LIN {X 0,Y 425.295,Z 309.51,A -85,B 0,C 180,E1 20716.386,E2 20716.386} C_VEL
LIN {X 0,Y 425.304,Z 309.491,A -85,B 0,C 180,E1 20712.629,E2 20712.629} C_VEL
LIN {X 0,Y 425.291,Z 309.491,A -85,B 0,C 180,E1 20708.79,E2 20708.79} C_VEL
LIN {X 0,Y 425.259,Z 309.512,A -85,B 0,C 180,E1 20705.126,E2 20705.126} C_VEL
LIN {X 0,Y 425.246,Z 309.506,A -85,B 0,C 180,E1 20701.347,E2 20701.347} C_VEL
LIN {X 0,Y 425.238,Z 309.495,A -85,B 0,C 180,E1 20697.574,E2 20697.574} C_VEL
LIN {X 0,Y 425.253,Z 309.511,A -85,B 0,C 180,E1 20693.791,E2 20693.791} C_VEL
LIN {X 0,Y 425.279,Z 309.498,A -85,B 0,C 180,E1 20690.086,E2 20690.086} C_VEL
LIN {X 0,Y 425.305,Z 309.487,A -85,B 0,C 180,E1 20686.264,E2 20686.264} C_VEL
LIN {X 0,Y 425.294,Z 309.508,A -85,B 0,C 180,E1 20682.486,E2 20682.486} C_VEL
LIN {X 0,Y 425.275,Z 309.503,A -85,B 0,C 180,E1 20678.772,E2 20678.772} C_VEL
LIN {X 0,Y 425.262,Z 309.492,A -85,B 0,C 180,E1 20675.111,E2 20675.111} C_VEL
LIN {X 0,Y 425.268,Z 309.502,A -85,B 0,C 180,E1 20671.276,E2 20671.276} C_VEL
LIN {X 0,Y 425.284,Z 309.507,A -85,B 0,C 180,E1 20667.565,E2 20667.565} C_VEL
LIN {X 0,Y 425.308,Z 309.508,A -85,B 0,C 180,E1 20663.837,E2 20663.837} C_VEL
LIN {X 0,Y 425.328,Z 309.506,A -85,B 0,C 180,E1 20660.026,E2 20660.026} C_VEL
LIN {X 0,Y 425.318,Z 309.499,A -85,B 0,C 180,E1 20656.092,E2 20656.092} C_VEL
LIN {X 0,Y 425.311,Z 309.478,A -85,B 0,C 180,E1 20652.223,E2 20652.223} C_VEL
LIN {X 0,Y 425.322,Z 309.731,A -85,B 0,C 180,E1 20648.704,E2 20648.704} C_VEL
LIN {X 0,Y 431.316,Z 325.075,A -85,B 0,C 180,E1 20645.907,E2 20645.907} C_VEL
LIN {X 0,Y 437.334,Z 341.625,A -85,B 0,C 180,E1 20643.199,E2 20643.199} C_VEL
LIN {X 0,Y 438.46,Z 344.163,A -85,B 0,C 180,E1 20642.946,E2 20642.946} C_VEL
LIN {X 0,Y 445.18,Z 356.721,A -85,B 0,C 180,E1 20642.081,E2 20642.081} C_VEL
LIN {X 0,Y 447.01,Z 366.68,A -85,B 0,C 180,E1 20641.733,E2 20641.733} C_VEL
LIN {X 0,Y 443.897,Z 554.794,A -85,B 0,C 180,E1 20638.73,E2 20638.73} C_VEL
LIN {X 0,Y 442.939,Z 562.472,A -85,B 0,C 180,E1 20638.628,E2 20638.628} C_VEL
LIN {X 0,Y 437.427,Z 580.609,A -85,B 0,C 180,E1 20638.46,E2 20638.46} C_VEL
LIN {X 0,Y 435.926,Z 588.027,A -85,B 0,C 180,E1 20638.239,E2 20638.239} C_VEL
LIN {X 0,Y 435.833,Z 589.062,A -85,B 0,C 180,E1 20638.193,E2 20638.193} C_VEL
LIN {X 0,Y 434.586,Z 606.139,A -85,B 0,C 180,E1 20637.321,E2 20637.321} C_VEL
LIN {X 0,Y 432.916,Z 623.479,A -85,B 0,C 180,E1 20636.175,E2 20636.175} C_VEL
LIN {X 0,Y 430.996,Z 639.731,A -85,B 0,C 180,E1 20634.827,E2 20634.827} C_VEL
LIN {X 0,Y 428.968,Z 654.603,A -85,B 0,C 180,E1 20633.313,E2 20633.313} C_VEL
LIN {X 0,Y 426.86,Z 668.614,A -85,B 0,C 180,E1 20631.576,E2 20631.576} C_VEL
LIN {X 0,Y 424.795,Z 681.338,A -85,B 0,C 180,E1 20629.668,E2 20629.668} C_VEL
LIN {X 0,Y 422.892,Z 692.644,A -85,B 0,C 180,E1 20627.615,E2 20627.615} C_VEL
LIN {X 0,Y 421.141,Z 703.114,A -85,B 0,C 180,E1 20625.279,E2 20625.279} C_VEL
LIN {X 0,Y 419.749,Z 711.572,A -85,B 0,C 180,E1 20622.939,E2 20622.939} C_VEL
LIN {X 0,Y 418.624,Z 718.946,A -85,B 0,C 180,E1 20620.319,E2 20620.319} C_VEL
LIN {X 0,Y 417.88,Z 724.436,A -85,B 0,C 180,E1 20617.7,E2 20617.7} C_VEL
LIN {X 0,Y 417.414,Z 728.221,A -85,B 0,C 180,E1 20615.085,E2 20615.085} C_VEL
LIN {X 0,Y 417.168,Z 730.486,A -85,B 0,C 180,E1 20612.335,E2 20612.335} C_VEL
LIN {X 0,Y 417.109,Z 731.085,A -85,B 0,C 180,E1 20609.588,E2 20609.588} C_VEL
LIN {X 0,Y 417.21,Z 730.043,A -85,B 0,C 180,E1 20606.84,E2 20606.84} C_VEL
LIN {X 0,Y 417.516,Z 727.312,A -85,B 0,C 180,E1 20604.09,E2 20604.09} C_VEL
LIN {X 0,Y 418.1,Z 722.784,A -85,B 0,C 180,E1 20601.335,E2 20601.335} C_VEL
LIN {X 0,Y 418.949,Z 716.685,A -85,B 0,C 180,E1 20598.715,E2 20598.715} C_VEL
LIN {X 0,Y 420.139,Z 709.085,A -85,B 0,C 180,E1 20596.233,E2 20596.233} C_VEL
LIN {X 0,Y 421.646,Z 700.029,A -85,B 0,C 180,E1 20593.893,E2 20593.893} C_VEL
LIN {X 0,Y 423.426,Z 689.42,A -85,B 0,C 180,E1 20591.672,E2 20591.672} C_VEL
LIN {X 0,Y 425.411,Z 677.603,A -85,B 0,C 180,E1 20589.645,E2 20589.645} C_VEL
LIN {X 0,Y 427.552,Z 664.114,A -85,B 0,C 180,E1 20587.738,E2 20587.738} C_VEL
LIN {X 0,Y 429.701,Z 649.518,A -85,B 0,C 180,E1 20586.045,E2 20586.045} C_VEL
LIN {X 0,Y 431.738,Z 633.856,A -85,B 0,C 180,E1 20584.559,E2 20584.559} C_VEL
LIN {X 0,Y 433.596,Z 617.11,A -85,B 0,C 180,E1 20583.279,E2 20583.279} C_VEL
LIN {X 0,Y 435.079,Z 600.265,A -85,B 0,C 180,E1 20582.26,E2 20582.26} C_VEL
LIN {X 0,Y 436.268,Z 581.748,A -85,B 0,C 180,E1 20581.409,E2 20581.409} C_VEL
LIN {X 0,Y 436.995,Z 563.024,A -85,B 0,C 180,E1 20580.806,E2 20580.806} C_VEL
LIN {X 0,Y 437.369,Z 538.708,A -85,B 0,C 180,E1 20580.338,E2 20580.338} C_VEL
LIN {X 0,Y 440.401,Z 366.683,A -85,B 0,C 180,E1 20577.558,E2 20577.558} C_VEL
LIN {X 0,Y 438.664,Z 359.169,A -85,B 0,C 180,E1 20577.254,E2 20577.254} C_VEL
LIN {X 0,Y 429.753,Z 342.969,A -85,B 0,C 180,E1 20576.041,E2 20576.041} C_VEL
LIN {X 0,Y 423.803,Z 326.84,A -85,B 0,C 180,E1 20573.336,E2 20573.336} C_VEL
LIN {X 0,Y 418.468,Z 313.652,A -85,B 0,C 180,E1 20570.893,E2 20570.893} C_VEL
LIN {X 0,Y 417.399,Z 310.595,A -85,B 0,C 180,E1 20570.241,E2 20570.241} C_VEL
LIN {X 0,Y 417.367,Z 310.446,A -85,B 0,C 180,E1 20566.343,E2 20566.343} C_VEL
LIN {X 0,Y 417.361,Z 310.494,A -85,B 0,C 180,E1 20562.452,E2 20562.452} C_VEL
LIN {X 0,Y 417.347,Z 310.491,A -85,B 0,C 180,E1 20558.649,E2 20558.649} C_VEL
LIN {X 0,Y 417.341,Z 310.491,A -85,B 0,C 180,E1 20554.764,E2 20554.764} C_VEL
LIN {X 0,Y 417.335,Z 310.495,A -85,B 0,C 180,E1 20550.845,E2 20550.845} C_VEL
LIN {X 0,Y 417.335,Z 310.499,A -85,B 0,C 180,E1 20546.924,E2 20546.924} C_VEL
LIN {X 0,Y 417.336,Z 310.498,A -85,B 0,C 180,E1 20543.079,E2 20543.079} C_VEL
LIN {X 0,Y 417.355,Z 310.477,A -85,B 0,C 180,E1 20539.451,E2 20539.451} C_VEL
LIN {X 0,Y 417.368,Z 310.483,A -85,B 0,C 180,E1 20535.564,E2 20535.564} C_VEL
LIN {X 0,Y 417.358,Z 310.496,A -85,B 0,C 180,E1 20531.75,E2 20531.75} C_VEL
LIN {X 0,Y 417.343,Z 310.478,A -85,B 0,C 180,E1 20527.849,E2 20527.849} C_VEL
LIN {X 0,Y 417.317,Z 310.49,A -85,B 0,C 180,E1 20524.122,E2 20524.122} C_VEL
LIN {X 0,Y 417.302,Z 310.501,A -85,B 0,C 180,E1 20520.412,E2 20520.412} C_VEL
LIN {X 0,Y 417.303,Z 310.484,A -85,B 0,C 180,E1 20516.566,E2 20516.566} C_VEL
LIN {X 0,Y 417.318,Z 310.487,A -85,B 0,C 180,E1 20512.843,E2 20512.843} C_VEL
LIN {X 0,Y 417.345,Z 310.499,A -85,B 0,C 180,E1 20509.09,E2 20509.09} C_VEL
LIN {X 0,Y 417.373,Z 310.483,A -85,B 0,C 180,E1 20505.29,E2 20505.29} C_VEL
LIN {X 0,Y 417.364,Z 310.479,A -85,B 0,C 180,E1 20501.421,E2 20501.421} C_VEL
LIN {X 0,Y 417.353,Z 310.485,A -85,B 0,C 180,E1 20497.61,E2 20497.61} C_VEL
LIN {X 0,Y 417.34,Z 310.493,A -85,B 0,C 180,E1 20493.844,E2 20493.844} C_VEL
LIN {X 0,Y 417.334,Z 310.497,A -85,B 0,C 180,E1 20490.111,E2 20490.111} C_VEL
LIN {X 0,Y 417.337,Z 310.486,A -85,B 0,C 180,E1 20486.233,E2 20486.233} C_VEL
LIN {X 0,Y 417.341,Z 310.465,A -85,B 0,C 180,E1 20482.344,E2 20482.344} C_VEL
LIN {X 0,Y 417.358,Z 310.451,A -85,B 0,C 180,E1 20478.608,E2 20478.608} C_VEL
LIN {X 0,Y 417.389,Z 310.785,A -85,B 0,C 180,E1 20478.001,E2 20478.001} C_VEL
LIN {X 0,Y 418.612,Z 313.856,A -85,B 0,C 180,E1 20477.472,E2 20477.472} C_VEL
LIN {X 0,Y 425.196,Z 327.627,A -85,B 0,C 180,E1 20475.324,E2 20475.324} C_VEL
LIN {X 0,Y 433.412,Z 346.345,A -85,B 0,C 180,E1 20472.705,E2 20472.705} C_VEL
LIN {X 0,Y 439.742,Z 362.777,A -85,B 0,C 180,E1 20470.648,E2 20470.648} C_VEL
LIN {X 0,Y 437.871,Z 383.994,A -85,B 0,C 180,E1 20469.058,E2 20469.058} C_VEL
LIN {X 0,Y 441.535,Z 419.357,A -85,B 0,C 180,E1 20467.995,E2 20467.995} C_VEL
LIN {X 0,Y 435.739,Z 636.384,A -85,B 0,C 180,E1 20464.015,E2 20464.015} C_VEL
LIN {X 0,Y 434.519,Z 657.893,A -85,B 0,C 180,E1 20463.442,E2 20463.442} C_VEL
LIN {X 0,Y 432.751,Z 679.3,A -85,B 0,C 180,E1 20462.622,E2 20462.622} C_VEL
LIN {X 0,Y 430.784,Z 699.969,A -85,B 0,C 180,E1 20461.559,E2 20461.559} C_VEL
LIN {X 0,Y 428.751,Z 719.018,A -85,B 0,C 180,E1 20460.323,E2 20460.323} C_VEL
LIN {X 0,Y 426.668,Z 737.44,A -85,B 0,C 180,E1 20458.864,E2 20458.864} C_VEL
LIN {X 0,Y 424.603,Z 755.114,A -85,B 0,C 180,E1 20457.182,E2 20457.182} C_VEL
LIN {X 0,Y 422.491,Z 773.079,A -85,B 0,C 180,E1 20455.137,E2 20455.137} C_VEL
LIN {X 0,Y 420.637,Z 789.749,A -85,B 0,C 180,E1 20452.869,E2 20452.869} C_VEL
LIN {X 0,Y 419.154,Z 804.214,A -85,B 0,C 180,E1 20450.527,E2 20450.527} C_VEL
LIN {X 0,Y 418.029,Z 816.771,A -85,B 0,C 180,E1 20448.115,E2 20448.115} C_VEL
LIN {X 0,Y 417.232,Z 827.882,A -85,B 0,C 180,E1 20445.568,E2 20445.568} C_VEL
LIN {X 0,Y 416.703,Z 837.456,A -85,B 0,C 180,E1 20442.894,E2 20442.894} C_VEL
LIN {X 0,Y 416.453,Z 845.052,A -85,B 0,C 180,E1 20440.234,E2 20440.234} C_VEL
LIN {X 0,Y 416.366,Z 850.572,A -85,B 0,C 180,E1 20437.728,E2 20437.728} C_VEL
LIN {X 0,Y 416.386,Z 854.593,A -85,B 0,C 180,E1 20435.097,E2 20435.097} C_VEL
LIN {X 0,Y 416.426,Z 856.966,A -85,B 0,C 180,E1 20432.477,E2 20432.477} C_VEL
LIN {X 0,Y 416.447,Z 857.743,A -85,B 0,C 180,E1 20429.862,E2 20429.862} C_VEL
LIN {X 0,Y 416.427,Z 856.813,A -85,B 0,C 180,E1 20427.248,E2 20427.248} C_VEL
LIN {X 0,Y 416.387,Z 854.237,A -85,B 0,C 180,E1 20424.627,E2 20424.627} C_VEL
LIN {X 0,Y 416.374,Z 850.01,A -85,B 0,C 180,E1 20421.994,E2 20421.994} C_VEL
LIN {X 0,Y 416.483,Z 844.036,A -85,B 0,C 180,E1 20419.348,E2 20419.348} C_VEL
LIN {X 0,Y 416.764,Z 836.113,A -85,B 0,C 180,E1 20416.685,E2 20416.685} C_VEL
LIN {X 0,Y 417.308,Z 826.752,A -85,B 0,C 180,E1 20414.149,E2 20414.149} C_VEL
LIN {X 0,Y 418.148,Z 815.386,A -85,B 0,C 180,E1 20411.602,E2 20411.602} C_VEL
LIN {X 0,Y 419.315,Z 802.509,A -85,B 0,C 180,E1 20409.183,E2 20409.183} C_VEL
LIN {X 0,Y 420.797,Z 788.255,A -85,B 0,C 180,E1 20406.918,E2 20406.918} C_VEL
LIN {X 0,Y 422.553,Z 772.476,A -85,B 0,C 180,E1 20404.792,E2 20404.792} C_VEL
LIN {X 0,Y 424.601,Z 755.097,A -85,B 0,C 180,E1 20402.818,E2 20402.818} C_VEL
LIN {X 0,Y 426.762,Z 736.64,A -85,B 0,C 180,E1 20401.067,E2 20401.067} C_VEL
LIN {X 0,Y 428.972,Z 717.108,A -85,B 0,C 180,E1 20399.54,E2 20399.54} C_VEL
LIN {X 0,Y 431.019,Z 697.589,A -85,B 0,C 180,E1 20398.304,E2 20398.304} C_VEL
LIN {X 0,Y 432.834,Z 678.286,A -85,B 0,C 180,E1 20397.335,E2 20397.335} C_VEL
LIN {X 0,Y 434.552,Z 657.279,A -85,B 0,C 180,E1 20396.541,E2 20396.541} C_VEL
LIN {X 0,Y 435.772,Z 635.074,A -85,B 0,C 180,E1 20395.961,E2 20395.961} C_VEL
LIN {X 0,Y 441.555,Z 417.909,A -85,B 0,C 180,E1 20391.983,E2 20391.983} C_VEL
LIN {X 0,Y 437.832,Z 382.808,A -85,B 0,C 180,E1 20390.888,E2 20390.888} C_VEL
LIN {X 0,Y 439.679,Z 362.43,A -85,B 0,C 180,E1 20389.323,E2 20389.323} C_VEL
LIN {X 0,Y 431.887,Z 342.744,A -85,B 0,C 180,E1 20386.824,E2 20386.824} C_VEL
LIN {X 0,Y 423.924,Z 324.867,A -85,B 0,C 180,E1 20384.278,E2 20384.278} C_VEL
LIN {X 0,Y 419.049,Z 314.463,A -85,B 0,C 180,E1 20382.658,E2 20382.658} C_VEL
LIN {X 0,Y 417.415,Z 310.928,A -85,B 0,C 180,E1 20382.052,E2 20382.052} C_VEL
LIN {X 0,Y 417.349,Z 310.452,A -85,B 0,C 180,E1 20381.576,E2 20381.576} C_VEL
LIN {X 0,Y 417.34,Z 310.47,A -85,B 0,C 180,E1 20377.83,E2 20377.83} C_VEL
LIN {X 0,Y 417.339,Z 310.481,A -85,B 0,C 180,E1 20373.932,E2 20373.932} C_VEL
LIN {X 0,Y 417.341,Z 310.495,A -85,B 0,C 180,E1 20370.047,E2 20370.047} C_VEL
LIN {X 0,Y 417.351,Z 310.49,A -85,B 0,C 180,E1 20366.309,E2 20366.309} C_VEL
LIN {X 0,Y 417.369,Z 310.482,A -85,B 0,C 180,E1 20362.538,E2 20362.538} C_VEL
LIN {X 0,Y 417.371,Z 310.479,A -85,B 0,C 180,E1 20358.724,E2 20358.724} C_VEL
LIN {X 0,Y 417.36,Z 310.488,A -85,B 0,C 180,E1 20354.853,E2 20354.853} C_VEL
LIN {X 0,Y 417.336,Z 310.499,A -85,B 0,C 180,E1 20351.05,E2 20351.05} C_VEL
LIN {X 0,Y 417.316,Z 310.489,A -85,B 0,C 180,E1 20347.295,E2 20347.295} C_VEL
LIN {X 0,Y 417.307,Z 310.487,A -85,B 0,C 180,E1 20343.571,E2 20343.571} C_VEL
LIN {X 0,Y 417.308,Z 310.502,A -85,B 0,C 180,E1 20339.725,E2 20339.725} C_VEL
LIN {X 0,Y 417.322,Z 310.486,A -85,B 0,C 180,E1 20336.016,E2 20336.016} C_VEL
LIN {X 0,Y 417.355,Z 310.478,A -85,B 0,C 180,E1 20332.29,E2 20332.29} C_VEL
LIN {X 0,Y 417.357,Z 310.5,A -85,B 0,C 180,E1 20328.39,E2 20328.39} C_VEL
LIN {X 0,Y 417.349,Z 310.483,A -85,B 0,C 180,E1 20324.578,E2 20324.578} C_VEL
LIN {X 0,Y 417.33,Z 310.482,A -85,B 0,C 180,E1 20320.838,E2 20320.838} C_VEL
LIN {X 0,Y 417.324,Z 310.5,A -85,B 0,C 180,E1 20317.161,E2 20317.161} C_VEL
LIN {X 0,Y 417.328,Z 310.499,A -85,B 0,C 180,E1 20313.229,E2 20313.229} C_VEL
LIN {X 0,Y 417.333,Z 310.494,A -85,B 0,C 180,E1 20309.325,E2 20309.325} C_VEL
LIN {X 0,Y 417.344,Z 310.488,A -85,B 0,C 180,E1 20305.499,E2 20305.499} C_VEL
LIN {X 0,Y 417.37,Z 310.484,A -85,B 0,C 180,E1 20301.789,E2 20301.789} C_VEL
LIN {X 0,Y 417.382,Z 310.485,A -85,B 0,C 180,E1 20297.953,E2 20297.953} C_VEL
LIN {X 0,Y 417.375,Z 310.446,A -85,B 0,C 180,E1 20294.054,E2 20294.054} C_VEL
LIN {X 0,Y 417.381,Z 310.473,A -85,B 0,C 180,E1 20290.12,E2 20290.12} C_VEL
LIN {X 0,Y 417.423,Z 310.821,A -85,B 0,C 180,E1 20289.56,E2 20289.56} C_VEL
LIN {X 0,Y 423.284,Z 325.515,A -85,B 0,C 180,E1 20286.796,E2 20286.796} C_VEL
LIN {X 0,Y 429.434,Z 342.168,A -85,B 0,C 180,E1 20283.971,E2 20283.971} C_VEL
LIN {X 0,Y 430.778,Z 344.992,A -85,B 0,C 180,E1 20283.685,E2 20283.685} C_VEL
LIN {X 0,Y 439.064,Z 360.282,A -85,B 0,C 180,E1 20282.586,E2 20282.586} C_VEL
LIN {X 0,Y 440.446,Z 368.261,A -85,B 0,C 180,E1 20282.307,E2 20282.307} C_VEL
LIN {X 0,Y 437.093,Z 558.617,A -85,B 0,C 180,E1 20279.21,E2 20279.21} C_VEL
LIN {X 0,Y 436.455,Z 577.921,A -85,B 0,C 180,E1 20278.644,E2 20278.644} C_VEL
LIN {X 0,Y 435.833,Z 589.062,A -85,B 0,C 180,E1 20278.193,E2 20278.193} C_VEL
LIN {X 0,Y 434.477,Z 596.631,A -85,B 0,C 180,E1 20277.912,E2 20277.912} C_VEL
LIN {X 0,Y 428.112,Z 614.037,A -85,B 0,C 180,E1 20277.327,E2 20277.327} C_VEL
LIN {X 0,Y 426.369,Z 620.792,A -85,B 0,C 180,E1 20276.95,E2 20276.95} C_VEL
LIN {X 0,Y 426.252,Z 621.745,A -85,B 0,C 180,E1 20276.885,E2 20276.885} C_VEL
LIN {X 0,Y 424.256,Z 638.214,A -85,B 0,C 180,E1 20275.548,E2 20275.548} C_VEL
LIN {X 0,Y 422.152,Z 653.265,A -85,B 0,C 180,E1 20274.04,E2 20274.04} C_VEL
LIN {X 0,Y 420.017,Z 666.865,A -85,B 0,C 180,E1 20272.388,E2 20272.388} C_VEL
LIN {X 0,Y 417.793,Z 680.072,A -85,B 0,C 180,E1 20270.45,E2 20270.45} C_VEL
LIN {X 0,Y 415.714,Z 691.783,A -85,B 0,C 180,E1 20268.365,E2 20268.365} C_VEL
LIN {X 0,Y 413.892,Z 702.067,A -85,B 0,C 180,E1 20266.129,E2 20266.129} C_VEL
LIN {X 0,Y 412.327,Z 710.951,A -85,B 0,C 180,E1 20263.747,E2 20263.747} C_VEL
LIN {X 0,Y 411.096,Z 718.401,A -85,B 0,C 180,E1 20261.22,E2 20261.22} C_VEL
LIN {X 0,Y 410.21,Z 724.366,A -85,B 0,C 180,E1 20258.55,E2 20258.55} C_VEL
LIN {X 0,Y 409.629,Z 728.578,A -85,B 0,C 180,E1 20255.884,E2 20255.884} C_VEL
LIN {X 0,Y 409.305,Z 731.277,A -85,B 0,C 180,E1 20253.081,E2 20253.081} C_VEL
LIN {X 0,Y 409.2,Z 732.293,A -85,B 0,C 180,E1 20250.28,E2 20250.28} C_VEL
LIN {X 0,Y 409.271,Z 731.67,A -85,B 0,C 180,E1 20247.48,E2 20247.48} C_VEL
LIN {X 0,Y 409.538,Z 729.386,A -85,B 0,C 180,E1 20244.677,E2 20244.677} C_VEL
LIN {X 0,Y 410.084,Z 725.347,A -85,B 0,C 180,E1 20241.871,E2 20241.871} C_VEL
LIN {X 0,Y 410.908,Z 719.743,A -85,B 0,C 180,E1 20239.201,E2 20239.201} C_VEL
LIN {X 0,Y 412.133,Z 712.22,A -85,B 0,C 180,E1 20236.532,E2 20236.532} C_VEL
LIN {X 0,Y 413.645,Z 703.643,A -85,B 0,C 180,E1 20234.149,E2 20234.149} C_VEL
LIN {X 0,Y 415.525,Z 692.986,A -85,B 0,C 180,E1 20231.772,E2 20231.772} C_VEL
LIN {X 0,Y 417.57,Z 681.528,A -85,B 0,C 180,E1 20229.685,E2 20229.685} C_VEL
LIN {X 0,Y 419.849,Z 668.093,A -85,B 0,C 180,E1 20227.677,E2 20227.677} C_VEL
LIN {X 0,Y 422.052,Z 654.11,A -85,B 0,C 180,E1 20225.954,E2 20225.954} C_VEL
LIN {X 0,Y 424.252,Z 638.461,A -85,B 0,C 180,E1 20224.377,E2 20224.377} C_VEL
LIN {X 0,Y 426.243,Z 622.169,A -85,B 0,C 180,E1 20223.049,E2 20223.049} C_VEL
LIN {X 0,Y 427.946,Z 604.675,A -85,B 0,C 180,E1 20221.916,E2 20221.916} C_VEL
LIN {X 0,Y 429.264,Z 586.618,A -85,B 0,C 180,E1 20221.022,E2 20221.022} C_VEL
LIN {X 0,Y 430.126,Z 567.98,A -85,B 0,C 180,E1 20220.359,E2 20220.359} C_VEL
LIN {X 0,Y 430.528,Z 548.32,A -85,B 0,C 180,E1 20219.919,E2 20219.919} C_VEL
LIN {X 0,Y 433.863,Z 368.04,A -85,B 0,C 180,E1 20216.96,E2 20216.96} C_VEL
LIN {X 0,Y 432.581,Z 362.846,A -85,B 0,C 180,E1 20216.736,E2 20216.736} C_VEL
LIN {X 0,Y 421.819,Z 343.427,A -85,B 0,C 180,E1 20215.218,E2 20215.218} C_VEL
LIN {X 0,Y 415.921,Z 327.808,A -85,B 0,C 180,E1 20212.496,E2 20212.496} C_VEL
LIN {X 0,Y 410.61,Z 314.728,A -85,B 0,C 180,E1 20209.996,E2 20209.996} C_VEL
LIN {X 0,Y 409.438,Z 311.625,A -85,B 0,C 180,E1 20209.307,E2 20209.307} C_VEL
LIN {X 0,Y 409.42,Z 311.437,A -85,B 0,C 180,E1 20205.488,E2 20205.488} C_VEL
LIN {X 0,Y 409.436,Z 311.472,A -85,B 0,C 180,E1 20201.624,E2 20201.624} C_VEL
LIN {X 0,Y 409.442,Z 311.47,A -85,B 0,C 180,E1 20197.803,E2 20197.803} C_VEL
LIN {X 0,Y 409.438,Z 311.468,A -85,B 0,C 180,E1 20193.834,E2 20193.834} C_VEL
LIN {X 0,Y 409.449,Z 311.466,A -85,B 0,C 180,E1 20189.879,E2 20189.879} C_VEL
LIN {X 0,Y 409.43,Z 311.474,A -85,B 0,C 180,E1 20185.921,E2 20185.921} C_VEL
LIN {X 0,Y 409.415,Z 311.487,A -85,B 0,C 180,E1 20182.092,E2 20182.092} C_VEL
LIN {X 0,Y 409.398,Z 311.479,A -85,B 0,C 180,E1 20178.217,E2 20178.217} C_VEL
LIN {X 0,Y 409.381,Z 311.466,A -85,B 0,C 180,E1 20174.426,E2 20174.426} C_VEL
LIN {X 0,Y 409.377,Z 311.487,A -85,B 0,C 180,E1 20170.555,E2 20170.555} C_VEL
LIN {X 0,Y 409.37,Z 311.489,A -85,B 0,C 180,E1 20166.592,E2 20166.592} C_VEL
LIN {X 0,Y 409.364,Z 311.468,A -85,B 0,C 180,E1 20162.64,E2 20162.64} C_VEL
LIN {X 0,Y 409.372,Z 311.482,A -85,B 0,C 180,E1 20158.881,E2 20158.881} C_VEL
LIN {X 0,Y 409.394,Z 311.487,A -85,B 0,C 180,E1 20155.097,E2 20155.097} C_VEL
LIN {X 0,Y 409.416,Z 311.465,A -85,B 0,C 180,E1 20151.291,E2 20151.291} C_VEL
LIN {X 0,Y 409.422,Z 311.467,A -85,B 0,C 180,E1 20147.304,E2 20147.304} C_VEL
LIN {X 0,Y 409.429,Z 311.483,A -85,B 0,C 180,E1 20143.398,E2 20143.398} C_VEL
LIN {X 0,Y 409.429,Z 311.486,A -85,B 0,C 180,E1 20139.411,E2 20139.411} C_VEL
LIN {X 0,Y 409.413,Z 311.481,A -85,B 0,C 180,E1 20135.624,E2 20135.624} C_VEL
LIN {X 0,Y 409.404,Z 311.479,A -85,B 0,C 180,E1 20131.838,E2 20131.838} C_VEL
LIN {X 0,Y 409.4,Z 311.482,A -85,B 0,C 180,E1 20127.997,E2 20127.997} C_VEL
LIN {X 0,Y 409.395,Z 311.433,A -85,B 0,C 180,E1 20124.116,E2 20124.116} C_VEL
LIN {X 0,Y 409.404,Z 311.469,A -85,B 0,C 180,E1 20120.219,E2 20120.219} C_VEL
LIN {X 0,Y 409.488,Z 311.753,A -85,B 0,C 180,E1 20118.979,E2 20118.979} C_VEL
LIN {X 0,Y 410.878,Z 315.161,A -85,B 0,C 180,E1 20118.369,E2 20118.369} C_VEL
LIN {X 0,Y 417.354,Z 328.537,A -85,B 0,C 180,E1 20116.183,E2 20116.183} C_VEL
LIN {X 0,Y 425.615,Z 347.272,A -85,B 0,C 180,E1 20113.456,E2 20113.456} C_VEL
LIN {X 0,Y 432.84,Z 365.718,A -85,B 0,C 180,E1 20111.063,E2 20111.063} C_VEL
LIN {X 0,Y 431.181,Z 383.563,A -85,B 0,C 180,E1 20109.707,E2 20109.707} C_VEL
LIN {X 0,Y 434.934,Z 420.487,A -85,B 0,C 180,E1 20108.574,E2 20108.574} C_VEL
LIN {X 0,Y 428.868,Z 635.975,A -85,B 0,C 180,E1 20104.566,E2 20104.566} C_VEL
LIN {X 0,Y 427.59,Z 657.284,A -85,B 0,C 180,E1 20103.986,E2 20103.986} C_VEL
LIN {X 0,Y 425.77,Z 678.267,A -85,B 0,C 180,E1 20103.172,E2 20103.172} C_VEL
LIN {X 0,Y 423.67,Z 699.069,A -85,B 0,C 180,E1 20102.088,E2 20102.088} C_VEL
LIN {X 0,Y 421.507,Z 718.264,A -85,B 0,C 180,E1 20100.821,E2 20100.821} C_VEL
LIN {X 0,Y 419.298,Z 736.613,A -85,B 0,C 180,E1 20099.342,E2 20099.342} C_VEL
LIN {X 0,Y 417.021,Z 754.9,A -85,B 0,C 180,E1 20097.563,E2 20097.563} C_VEL
LIN {X 0,Y 414.87,Z 772.149,A -85,B 0,C 180,E1 20095.556,E2 20095.556} C_VEL
LIN {X 0,Y 412.957,Z 788.311,A -85,B 0,C 180,E1 20093.315,E2 20093.315} C_VEL
LIN {X 0,Y 411.362,Z 802.783,A -85,B 0,C 180,E1 20090.934,E2 20090.934} C_VEL
LIN {X 0,Y 410.167,Z 815.378,A -85,B 0,C 180,E1 20088.475,E2 20088.475} C_VEL
LIN {X 0,Y 409.313,Z 826.523,A -85,B 0,C 180,E1 20085.878,E2 20085.878} C_VEL
LIN {X 0,Y 408.754,Z 836.131,A -85,B 0,C 180,E1 20083.149,E2 20083.149} C_VEL
LIN {X 0,Y 408.506,Z 843.761,A -85,B 0,C 180,E1 20080.435,E2 20080.435} C_VEL
LIN {X 0,Y 408.424,Z 849.304,A -85,B 0,C 180,E1 20077.879,E2 20077.879} C_VEL
LIN {X 0,Y 408.46,Z 853.36,A -85,B 0,C 180,E1 20075.196,E2 20075.196} C_VEL
LIN {X 0,Y 408.514,Z 855.759,A -85,B 0,C 180,E1 20072.525,E2 20072.525} C_VEL
LIN {X 0,Y 408.54,Z 856.558,A -85,B 0,C 180,E1 20070,E2 20070} C_VEL
LIN {X 0,Y 408.515,Z 855.681,A -85,B 0,C 180,E1 20067.335,E2 20067.335} C_VEL
LIN {X 0,Y 408.462,Z 853.181,A -85,B 0,C 180,E1 20064.663,E2 20064.663} C_VEL
LIN {X 0,Y 408.429,Z 849.023,A -85,B 0,C 180,E1 20061.979,E2 20061.979} C_VEL
LIN {X 0,Y 408.516,Z 843.427,A -85,B 0,C 180,E1 20059.423,E2 20059.423} C_VEL
LIN {X 0,Y 408.765,Z 835.93,A -85,B 0,C 180,E1 20056.786,E2 20056.786} C_VEL
LIN {X 0,Y 409.313,Z 826.523,A -85,B 0,C 180,E1 20054.122,E2 20054.122} C_VEL
LIN {X 0,Y 410.167,Z 815.376,A -85,B 0,C 180,E1 20051.525,E2 20051.525} C_VEL
LIN {X 0,Y 411.364,Z 802.779,A -85,B 0,C 180,E1 20049.066,E2 20049.066} C_VEL
LIN {X 0,Y 412.956,Z 788.304,A -85,B 0,C 180,E1 20046.685,E2 20046.685} C_VEL
LIN {X 0,Y 414.868,Z 772.131,A -85,B 0,C 180,E1 20044.444,E2 20044.444} C_VEL
LIN {X 0,Y 417.103,Z 754.217,A -85,B 0,C 180,E1 20042.365,E2 20042.365} C_VEL
LIN {X 0,Y 419.395,Z 735.81,A -85,B 0,C 180,E1 20040.587,E2 20040.587} C_VEL
LIN {X 0,Y 421.736,Z 716.344,A -85,B 0,C 180,E1 20039.039,E2 20039.039} C_VEL
LIN {X 0,Y 423.888,Z 696.913,A -85,B 0,C 180,E1 20037.787,E2 20037.787} C_VEL
LIN {X 0,Y 425.839,Z 677.437,A -85,B 0,C 180,E1 20036.794,E2 20036.794} C_VEL
LIN {X 0,Y 427.644,Z 656.33,A -85,B 0,C 180,E1 20035.986,E2 20035.986} C_VEL
LIN {X 0,Y 428.917,Z 634.217,A -85,B 0,C 180,E1 20035.401,E2 20035.401} C_VEL
LIN {X 0,Y 434.949,Z 419.079,A -85,B 0,C 180,E1 20031.405,E2 20031.405} C_VEL
LIN {X 0,Y 431.128,Z 382.442,A -85,B 0,C 180,E1 20030.245,E2 20030.245} C_VEL
LIN {X 0,Y 432.662,Z 365.234,A -85,B 0,C 180,E1 20028.883,E2 20028.883} C_VEL
LIN {X 0,Y 424.953,Z 345.751,A -85,B 0,C 180,E1 20026.344,E2 20026.344} C_VEL
LIN {X 0,Y 416.913,Z 327.6,A -85,B 0,C 180,E1 20023.685,E2 20023.685} C_VEL
LIN {X 0,Y 410.84,Z 315.109,A -85,B 0,C 180,E1 20021.636,E2 20021.636} C_VEL
LIN {X 0,Y 409.479,Z 311.692,A -85,B 0,C 180,E1 20021.019,E2 20021.019} C_VEL
LIN {X 0,Y 409.431,Z 311.437,A -85,B 0,C 180,E1 20017.098,E2 20017.098} C_VEL
LIN {X 0,Y 409.427,Z 311.484,A -85,B 0,C 180,E1 20013.163,E2 20013.163} C_VEL
LIN {X 0,Y 409.412,Z 311.489,A -85,B 0,C 180,E1 20009.328,E2 20009.328} C_VEL
LIN {X 0,Y 409.395,Z 311.49,A -85,B 0,C 180,E1 20005.612,E2 20005.612} C_VEL
LIN {X 0,Y 409.389,Z 311.485,A -85,B 0,C 180,E1 20001.791,E2 20001.791} C_VEL
LIN {X 0,Y 409.389,Z 311.474,A -85,B 0,C 180,E1 19997.922,E2 19997.922} C_VEL
LIN {X 0,Y 409.395,Z 311.468,A -85,B 0,C 180,E1 19994.136,E2 19994.136} C_VEL
LIN {X 0,Y 409.405,Z 311.484,A -85,B 0,C 180,E1 19990.269,E2 19990.269} C_VEL
LIN {X 0,Y 409.423,Z 311.48,A -85,B 0,C 180,E1 19986.45,E2 19986.45} C_VEL
LIN {X 0,Y 409.413,Z 311.464,A -85,B 0,C 180,E1 19982.519,E2 19982.519} C_VEL
LIN {X 0,Y 409.397,Z 311.481,A -85,B 0,C 180,E1 19978.74,E2 19978.74} C_VEL
LIN {X 0,Y 409.389,Z 311.486,A -85,B 0,C 180,E1 19974.815,E2 19974.815} C_VEL
LIN {X 0,Y 409.37,Z 311.466,A -85,B 0,C 180,E1 19971.148,E2 19971.148} C_VEL
LIN {X 0,Y 409.372,Z 311.487,A -85,B 0,C 180,E1 19967.301,E2 19967.301} C_VEL
LIN {X 0,Y 409.38,Z 311.488,A -85,B 0,C 180,E1 19963.396,E2 19963.396} C_VEL
LIN {X 0,Y 409.386,Z 311.473,A -85,B 0,C 180,E1 19959.558,E2 19959.558} C_VEL
LIN {X 0,Y 409.415,Z 311.468,A -85,B 0,C 180,E1 19955.93,E2 19955.93} C_VEL
LIN {X 0,Y 409.434,Z 311.48,A -85,B 0,C 180,E1 19952.038,E2 19952.038} C_VEL
LIN {X 0,Y 409.442,Z 311.486,A -85,B 0,C 180,E1 19948.165,E2 19948.165} C_VEL
LIN {X 0,Y 409.438,Z 311.488,A -85,B 0,C 180,E1 19944.167,E2 19944.167} C_VEL
LIN {X 0,Y 409.441,Z 311.487,A -85,B 0,C 180,E1 19940.222,E2 19940.222} C_VEL
LIN {X 0,Y 409.432,Z 311.48,A -85,B 0,C 180,E1 19936.282,E2 19936.282} C_VEL
LIN {X 0,Y 409.423,Z 311.449,A -85,B 0,C 180,E1 19932.377,E2 19932.377} C_VEL
LIN {X 0,Y 409.445,Z 311.68,A -85,B 0,C 180,E1 19930.554,E2 19930.554} C_VEL
LIN {X 0,Y 414.039,Z 322.964,A -85,B 0,C 180,E1 19928.294,E2 19928.294} C_VEL
LIN {X 0,Y 420.183,Z 338.961,A -85,B 0,C 180,E1 19925.412,E2 19925.412} C_VEL
LIN {X 0,Y 422.114,Z 344.155,A -85,B 0,C 180,E1 19924.601,E2 19924.601} C_VEL
LIN {X 0,Y 432.944,Z 363.641,A -85,B 0,C 180,E1 19923.111,E2 19923.111} C_VEL
LIN {X 0,Y 433.926,Z 369.853,A -85,B 0,C 180,E1 19922.897,E2 19922.897} C_VEL
LIN {X 0,Y 430.344,Z 559.389,A -85,B 0,C 180,E1 19919.769,E2 19919.769} C_VEL
LIN {X 0,Y 429.672,Z 578.718,A -85,B 0,C 180,E1 19919.195,E2 19919.195} C_VEL
LIN {X 0,Y 428.534,Z 597.005,A -85,B 0,C 180,E1 19918.403,E2 19918.403} C_VEL
LIN {X 0,Y 427.032,Z 614.436,A -85,B 0,C 180,E1 19917.392,E2 19917.392} C_VEL
LIN {X 0,Y 426.252,Z 621.745,A -85,B 0,C 180,E1 19916.885,E2 19916.885} C_VEL
LIN {X 0,Y 424.656,Z 628.618,A -85,B 0,C 180,E1 19916.446,E2 19916.446} C_VEL
LIN {X 0,Y 417.575,Z 644.654,A -85,B 0,C 180,E1 19915.446,E2 19915.446} C_VEL
LIN {X 0,Y 415.555,Z 650.949,A -85,B 0,C 180,E1 19914.887,E2 19914.887} C_VEL
LIN {X 0,Y 415.401,Z 651.806,A -85,B 0,C 180,E1 19914.795,E2 19914.795} C_VEL
LIN {X 0,Y 412.991,Z 666.63,A -85,B 0,C 180,E1 19913.016,E2 19913.016} C_VEL
LIN {X 0,Y 410.554,Z 680.506,A -85,B 0,C 180,E1 19910.977,E2 19910.977} C_VEL
LIN {X 0,Y 408.344,Z 692.341,A -85,B 0,C 180,E1 19908.857,E2 19908.857} C_VEL
LIN {X 0,Y 406.394,Z 702.736,A -85,B 0,C 180,E1 19906.582,E2 19906.582} C_VEL
LIN {X 0,Y 404.717,Z 711.718,A -85,B 0,C 180,E1 19904.157,E2 19904.157} C_VEL
LIN {X 0,Y 403.38,Z 719.26,A -85,B 0,C 180,E1 19901.582,E2 19901.582} C_VEL
LIN {X 0,Y 402.414,Z 725.309,A -85,B 0,C 180,E1 19898.861,E2 19898.861} C_VEL
LIN {X 0,Y 401.778,Z 729.602,A -85,B 0,C 180,E1 19896.143,E2 19896.143} C_VEL
LIN {X 0,Y 401.414,Z 732.379,A -85,B 0,C 180,E1 19893.284,E2 19893.284} C_VEL
LIN {X 0,Y 401.291,Z 733.474,A -85,B 0,C 180,E1 19890.428,E2 19890.428} C_VEL
LIN {X 0,Y 401.356,Z 732.933,A -85,B 0,C 180,E1 19887.573,E2 19887.573} C_VEL
LIN {X 0,Y 401.632,Z 730.734,A -85,B 0,C 180,E1 19884.715,E2 19884.715} C_VEL
LIN {X 0,Y 402.161,Z 727.017,A -85,B 0,C 180,E1 19881.997,E2 19881.997} C_VEL
LIN {X 0,Y 403.008,Z 721.566,A -85,B 0,C 180,E1 19879.258,E2 19879.258} C_VEL
LIN {X 0,Y 404.18,Z 714.745,A -85,B 0,C 180,E1 19876.7,E2 19876.7} C_VEL
LIN {X 0,Y 405.709,Z 706.499,A -85,B 0,C 180,E1 19874.271,E2 19874.271} C_VEL
LIN {X 0,Y 407.496,Z 696.925,A -85,B 0,C 180,E1 19871.992,E2 19871.992} C_VEL
LIN {X 0,Y 409.545,Z 686.041,A -85,B 0,C 180,E1 19869.866,E2 19869.866} C_VEL
LIN {X 0,Y 411.773,Z 673.823,A -85,B 0,C 180,E1 19867.892,E2 19867.892} C_VEL
LIN {X 0,Y 414.185,Z 659.608,A -85,B 0,C 180,E1 19865.999,E2 19865.999} C_VEL
LIN {X 0,Y 416.559,Z 644.23,A -85,B 0,C 180,E1 19864.327,E2 19864.327} C_VEL
LIN {X 0,Y 418.648,Z 628.546,A -85,B 0,C 180,E1 19862.938,E2 19862.938} C_VEL
LIN {X 0,Y 420.602,Z 610.906,A -85,B 0,C 180,E1 19861.69,E2 19861.69} C_VEL
LIN {X 0,Y 422.101,Z 593.095,A -85,B 0,C 180,E1 19860.716,E2 19860.716} C_VEL
LIN {X 0,Y 423.186,Z 574.271,A -85,B 0,C 180,E1 19859.962,E2 19859.962} C_VEL
LIN {X 0,Y 423.733,Z 555.053,A -85,B 0,C 180,E1 19859.452,E2 19859.452} C_VEL
LIN {X 0,Y 427.381,Z 369.434,A -85,B 0,C 180,E1 19856.345,E2 19856.345} C_VEL
LIN {X 0,Y 426.448,Z 366.302,A -85,B 0,C 180,E1 19856.189,E2 19856.189} C_VEL
LIN {X 0,Y 414.197,Z 344.558,A -85,B 0,C 180,E1 19854.441,E2 19854.441} C_VEL
LIN {X 0,Y 408.67,Z 330.049,A -85,B 0,C 180,E1 19851.868,E2 19851.868} C_VEL
LIN {X 0,Y 402.76,Z 315.929,A -85,B 0,C 180,E1 19849.053,E2 19849.053} C_VEL
LIN {X 0,Y 401.525,Z 312.649,A -85,B 0,C 180,E1 19848.329,E2 19848.329} C_VEL
LIN {X 0,Y 401.478,Z 312.44,A -85,B 0,C 180,E1 19844.582,E2 19844.582} C_VEL
LIN {X 0,Y 401.468,Z 312.467,A -85,B 0,C 180,E1 19840.732,E2 19840.732} C_VEL
LIN {X 0,Y 401.464,Z 312.469,A -85,B 0,C 180,E1 19836.886,E2 19836.886} C_VEL
LIN {X 0,Y 401.46,Z 312.468,A -85,B 0,C 180,E1 19832.884,E2 19832.884} C_VEL
LIN {X 0,Y 401.461,Z 312.46,A -85,B 0,C 180,E1 19829.055,E2 19829.055} C_VEL
LIN {X 0,Y 401.464,Z 312.456,A -85,B 0,C 180,E1 19825.207,E2 19825.207} C_VEL
LIN {X 0,Y 401.472,Z 312.47,A -85,B 0,C 180,E1 19821.322,E2 19821.322} C_VEL
LIN {X 0,Y 401.475,Z 312.475,A -85,B 0,C 180,E1 19817.389,E2 19817.389} C_VEL
LIN {X 0,Y 401.485,Z 312.452,A -85,B 0,C 180,E1 19813.539,E2 19813.539} C_VEL
LIN {X 0,Y 401.478,Z 312.454,A -85,B 0,C 180,E1 19809.534,E2 19809.534} C_VEL
LIN {X 0,Y 401.473,Z 312.478,A -85,B 0,C 180,E1 19805.718,E2 19805.718} C_VEL
LIN {X 0,Y 401.463,Z 312.459,A -85,B 0,C 180,E1 19801.713,E2 19801.713} C_VEL
LIN {X 0,Y 401.446,Z 312.457,A -85,B 0,C 180,E1 19797.859,E2 19797.859} C_VEL
LIN {X 0,Y 401.445,Z 312.478,A -85,B 0,C 180,E1 19793.996,E2 19793.996} C_VEL
LIN {X 0,Y 401.44,Z 312.473,A -85,B 0,C 180,E1 19790.105,E2 19790.105} C_VEL
LIN {X 0,Y 401.439,Z 312.456,A -85,B 0,C 180,E1 19786.249,E2 19786.249} C_VEL
LIN {X 0,Y 401.443,Z 312.465,A -85,B 0,C 180,E1 19782.311,E2 19782.311} C_VEL
LIN {X 0,Y 401.45,Z 312.476,A -85,B 0,C 180,E1 19778.37,E2 19778.37} C_VEL
LIN {X 0,Y 401.457,Z 312.477,A -85,B 0,C 180,E1 19774.478,E2 19774.478} C_VEL
LIN {X 0,Y 401.472,Z 312.476,A -85,B 0,C 180,E1 19770.619,E2 19770.619} C_VEL
LIN {X 0,Y 401.482,Z 312.473,A -85,B 0,C 180,E1 19766.778,E2 19766.778} C_VEL
LIN {X 0,Y 401.487,Z 312.424,A -85,B 0,C 180,E1 19762.835,E2 19762.835} C_VEL
LIN {X 0,Y 401.483,Z 312.6,A -85,B 0,C 180,E1 19760.087,E2 19760.087} C_VEL
LIN {X 0,Y 401.977,Z 314.409,A -85,B 0,C 180,E1 19759.706,E2 19759.706} C_VEL
LIN {X 0,Y 403.647,Z 317.225,A -85,B 0,C 180,E1 19759.161,E2 19759.161} C_VEL
LIN {X 0,Y 411.959,Z 334.831,A -85,B 0,C 180,E1 19756.234,E2 19756.234} C_VEL
LIN {X 0,Y 419.94,Z 353.216,A -85,B 0,C 180,E1 19753.531,E2 19753.531} C_VEL
LIN {X 0,Y 425.942,Z 368.781,A -85,B 0,C 180,E1 19751.484,E2 19751.484} C_VEL
LIN {X 0,Y 424.548,Z 383.134,A -85,B 0,C 180,E1 19750.377,E2 19750.377} C_VEL
LIN {X 0,Y 428.378,Z 421.614,A -85,B 0,C 180,E1 19749.171,E2 19749.171} C_VEL
LIN {X 0,Y 422.044,Z 635.504,A -85,B 0,C 180,E1 19745.136,E2 19745.136} C_VEL
LIN {X 0,Y 420.703,Z 656.691,A -85,B 0,C 180,E1 19744.549,E2 19744.549} C_VEL
LIN {X 0,Y 418.852,Z 677.103,A -85,B 0,C 180,E1 19743.746,E2 19743.746} C_VEL
LIN {X 0,Y 416.672,Z 697.503,A -85,B 0,C 180,E1 19742.677,E2 19742.677} C_VEL
LIN {X 0,Y 414.42,Z 716.6,A -85,B 0,C 180,E1 19741.407,E2 19741.407} C_VEL
LIN {X 0,Y 412.063,Z 735.036,A -85,B 0,C 180,E1 19739.909,E2 19739.909} C_VEL
LIN {X 0,Y 409.64,Z 753.382,A -85,B 0,C 180,E1 19738.103,E2 19738.103} C_VEL
LIN {X 0,Y 407.343,Z 770.726,A -85,B 0,C 180,E1 19736.055,E2 19736.055} C_VEL
LIN {X 0,Y 405.274,Z 787.072,A -85,B 0,C 180,E1 19733.752,E2 19733.752} C_VEL
LIN {X 0,Y 403.568,Z 801.573,A -85,B 0,C 180,E1 19731.322,E2 19731.322} C_VEL
LIN {X 0,Y 402.31,Z 814.007,A -85,B 0,C 180,E1 19728.849,E2 19728.849} C_VEL
LIN {X 0,Y 401.391,Z 825.185,A -85,B 0,C 180,E1 19726.199,E2 19726.199} C_VEL
LIN {X 0,Y 400.807,Z 834.827,A -85,B 0,C 180,E1 19723.414,E2 19723.414} C_VEL
LIN {X 0,Y 400.554,Z 842.489,A -85,B 0,C 180,E1 19720.644,E2 19720.644} C_VEL
LIN {X 0,Y 400.48,Z 848.054,A -85,B 0,C 180,E1 19718.037,E2 19718.037} C_VEL
LIN {X 0,Y 400.534,Z 852.136,A -85,B 0,C 180,E1 19715.299,E2 19715.299} C_VEL
LIN {X 0,Y 400.6,Z 854.552,A -85,B 0,C 180,E1 19712.575,E2 19712.575} C_VEL
LIN {X 0,Y 400.631,Z 855.357,A -85,B 0,C 180,E1 19710,E2 19710} C_VEL
LIN {X 0,Y 400.601,Z 854.551,A -85,B 0,C 180,E1 19707.425,E2 19707.425} C_VEL
LIN {X 0,Y 400.534,Z 852.135,A -85,B 0,C 180,E1 19704.701,E2 19704.701} C_VEL
LIN {X 0,Y 400.481,Z 848.055,A -85,B 0,C 180,E1 19701.963,E2 19701.963} C_VEL
LIN {X 0,Y 400.554,Z 842.493,A -85,B 0,C 180,E1 19699.356,E2 19699.356} C_VEL
LIN {X 0,Y 400.808,Z 834.829,A -85,B 0,C 180,E1 19696.586,E2 19696.586} C_VEL
LIN {X 0,Y 401.392,Z 825.183,A -85,B 0,C 180,E1 19693.801,E2 19693.801} C_VEL
LIN {X 0,Y 402.31,Z 814.003,A -85,B 0,C 180,E1 19691.151,E2 19691.151} C_VEL
LIN {X 0,Y 403.587,Z 801.368,A -85,B 0,C 180,E1 19688.643,E2 19688.643} C_VEL
LIN {X 0,Y 405.27,Z 787.067,A -85,B 0,C 180,E1 19686.249,E2 19686.249} C_VEL
LIN {X 0,Y 407.34,Z 770.711,A -85,B 0,C 180,E1 19683.946,E2 19683.946} C_VEL
LIN {X 0,Y 409.638,Z 753.353,A -85,B 0,C 180,E1 19681.896,E2 19681.896} C_VEL
LIN {X 0,Y 412.059,Z 734.996,A -85,B 0,C 180,E1 19680.091,E2 19680.091} C_VEL
LIN {X 0,Y 414.537,Z 715.605,A -85,B 0,C 180,E1 19678.521,E2 19678.521} C_VEL
LIN {X 0,Y 416.797,Z 696.261,A -85,B 0,C 180,E1 19677.252,E2 19677.252} C_VEL
LIN {X 0,Y 418.842,Z 677.041,A -85,B 0,C 180,E1 19676.255,E2 19676.255} C_VEL
LIN {X 0,Y 420.754,Z 655.774,A -85,B 0,C 180,E1 19675.425,E2 19675.425} C_VEL
LIN {X 0,Y 422.094,Z 633.713,A -85,B 0,C 180,E1 19674.83,E2 19674.83} C_VEL
LIN {X 0,Y 428.393,Z 420.171,A -85,B 0,C 180,E1 19670.807,E2 19670.807} C_VEL
LIN {X 0,Y 424.501,Z 381.848,A -85,B 0,C 180,E1 19669.564,E2 19669.564} C_VEL
LIN {X 0,Y 425.87,Z 368.617,A -85,B 0,C 180,E1 19668.499,E2 19668.499} C_VEL
LIN {X 0,Y 418.455,Z 349.723,A -85,B 0,C 180,E1 19665.989,E2 19665.989} C_VEL
LIN {X 0,Y 410.699,Z 332.17,A -85,B 0,C 180,E1 19663.356,E2 19663.356} C_VEL
LIN {X 0,Y 404.68,Z 319.763,A -85,B 0,C 180,E1 19661.276,E2 19661.276} C_VEL
LIN {X 0,Y 403.187,Z 316.439,A -85,B 0,C 180,E1 19660.708,E2 19660.708} C_VEL
LIN {X 0,Y 401.523,Z 312.834,A -85,B 0,C 180,E1 19660.034,E2 19660.034} C_VEL
LIN {X 0,Y 401.471,Z 312.461,A -85,B 0,C 180,E1 19659.61,E2 19659.61} C_VEL
LIN {X 0,Y 401.458,Z 312.421,A -85,B 0,C 180,E1 19655.718,E2 19655.718} C_VEL
LIN {X 0,Y 401.461,Z 312.469,A -85,B 0,C 180,E1 19651.869,E2 19651.869} C_VEL
LIN {X 0,Y 401.458,Z 312.467,A -85,B 0,C 180,E1 19647.919,E2 19647.919} C_VEL
LIN {X 0,Y 401.457,Z 312.468,A -85,B 0,C 180,E1 19643.951,E2 19643.951} C_VEL
LIN {X 0,Y 401.459,Z 312.474,A -85,B 0,C 180,E1 19640.102,E2 19640.102} C_VEL
LIN {X 0,Y 401.463,Z 312.479,A -85,B 0,C 180,E1 19636.197,E2 19636.197} C_VEL
LIN {X 0,Y 401.472,Z 312.461,A -85,B 0,C 180,E1 19632.367,E2 19632.367} C_VEL
LIN {X 0,Y 401.48,Z 312.452,A -85,B 0,C 180,E1 19628.449,E2 19628.449} C_VEL
LIN {X 0,Y 401.476,Z 312.469,A -85,B 0,C 180,E1 19624.571,E2 19624.571} C_VEL
LIN {X 0,Y 401.482,Z 312.471,A -85,B 0,C 180,E1 19620.57,E2 19620.57} C_VEL
LIN {X 0,Y 401.462,Z 312.453,A -85,B 0,C 180,E1 19616.536,E2 19616.536} C_VEL
LIN {X 0,Y 401.471,Z 312.459,A -85,B 0,C 180,E1 19612.559,E2 19612.559} C_VEL
LIN {X 0,Y 401.463,Z 312.478,A -85,B 0,C 180,E1 19608.653,E2 19608.653} C_VEL
LIN {X 0,Y 401.448,Z 312.459,A -85,B 0,C 180,E1 19604.84,E2 19604.84} C_VEL
LIN {X 0,Y 401.448,Z 312.46,A -85,B 0,C 180,E1 19600.957,E2 19600.957} C_VEL
LIN {X 0,Y 401.447,Z 312.478,A -85,B 0,C 180,E1 19597.136,E2 19597.136} C_VEL
LIN {X 0,Y 401.451,Z 312.477,A -85,B 0,C 180,E1 19593.205,E2 19593.205} C_VEL
LIN {X 0,Y 401.454,Z 312.472,A -85,B 0,C 180,E1 19589.23,E2 19589.23} C_VEL
LIN {X 0,Y 401.459,Z 312.467,A -85,B 0,C 180,E1 19585.272,E2 19585.272} C_VEL
LIN {X 0,Y 401.469,Z 312.466,A -85,B 0,C 180,E1 19581.444,E2 19581.444} C_VEL
LIN {X 0,Y 401.489,Z 312.466,A -85,B 0,C 180,E1 19577.699,E2 19577.699} C_VEL
LIN {X 0,Y 401.491,Z 312.42,A -85,B 0,C 180,E1 19573.763,E2 19573.763} C_VEL
LIN {X 0,Y 401.525,Z 312.728,A -85,B 0,C 180,E1 19571.528,E2 19571.528} C_VEL
LIN {X 0,Y 402.853,Z 316.073,A -85,B 0,C 180,E1 19570.8,E2 19570.8} C_VEL
LIN {X 0,Y 408.845,Z 330.583,A -85,B 0,C 180,E1 19567.924,E2 19567.924} C_VEL
LIN {X 0,Y 414.239,Z 344.647,A -85,B 0,C 180,E1 19565.449,E2 19565.449} C_VEL
LIN {X 0,Y 426.584,Z 366.634,A -85,B 0,C 180,E1 19563.687,E2 19563.687} C_VEL
LIN {X 0,Y 427.461,Z 371.054,A -85,B 0,C 180,E1 19563.512,E2 19563.512} C_VEL
LIN {X 0,Y 423.636,Z 560.134,A -85,B 0,C 180,E1 19560.345,E2 19560.345} C_VEL
LIN {X 0,Y 422.93,Z 579.467,A -85,B 0,C 180,E1 19559.765,E2 19559.765} C_VEL
LIN {X 0,Y 421.763,Z 597.411,A -85,B 0,C 180,E1 19558.981,E2 19558.981} C_VEL
LIN {X 0,Y 420.184,Z 615,A -85,B 0,C 180,E1 19557.954,E2 19557.954} C_VEL
LIN {X 0,Y 418.23,Z 631.776,A -85,B 0,C 180,E1 19556.708,E2 19556.708} C_VEL
LIN {X 0,Y 416.059,Z 647.549,A -85,B 0,C 180,E1 19555.249,E2 19555.249} C_VEL
LIN {X 0,Y 415.401,Z 651.806,A -85,B 0,C 180,E1 19554.795,E2 19554.795} C_VEL
LIN {X 0,Y 413.589,Z 657.941,A -85,B 0,C 180,E1 19554.181,E2 19554.181} C_VEL
LIN {X 0,Y 406.154,Z 672.262,A -85,B 0,C 180,E1 19552.777,E2 19552.777} C_VEL
LIN {X 0,Y 404.023,Z 677.673,A -85,B 0,C 180,E1 19552.053,E2 19552.053} C_VEL
LIN {X 0,Y 403.855,Z 678.401,A -85,B 0,C 180,E1 19551.937,E2 19551.937} C_VEL
LIN {X 0,Y 401.456,Z 690.73,A -85,B 0,C 180,E1 19549.798,E2 19549.798} C_VEL
LIN {X 0,Y 399.286,Z 701.631,A -85,B 0,C 180,E1 19547.487,E2 19547.487} C_VEL
LIN {X 0,Y 397.364,Z 711.344,A -85,B 0,C 180,E1 19544.931,E2 19544.931} C_VEL
LIN {X 0,Y 395.898,Z 719.007,A -85,B 0,C 180,E1 19542.396,E2 19542.396} C_VEL
LIN {X 0,Y 394.773,Z 725.428,A -85,B 0,C 180,E1 19539.623,E2 19539.623} C_VEL
LIN {X 0,Y 394.021,Z 730.07,A -85,B 0,C 180,E1 19536.85,E2 19536.85} C_VEL
LIN {X 0,Y 393.572,Z 733.178,A -85,B 0,C 180,E1 19533.933,E2 19533.933} C_VEL
LIN {X 0,Y 393.392,Z 734.595,A -85,B 0,C 180,E1 19531.019,E2 19531.019} C_VEL
LIN {X 0,Y 393.423,Z 734.376,A -85,B 0,C 180,E1 19528.107,E2 19528.107} C_VEL
LIN {X 0,Y 393.666,Z 732.51,A -85,B 0,C 180,E1 19525.192,E2 19525.192} C_VEL
LIN {X 0,Y 394.166,Z 729.146,A -85,B 0,C 180,E1 19522.421,E2 19522.421} C_VEL
LIN {X 0,Y 394.99,Z 724.109,A -85,B 0,C 180,E1 19519.647,E2 19519.647} C_VEL
LIN {X 0,Y 396.186,Z 717.445,A -85,B 0,C 180,E1 19516.946,E2 19516.946} C_VEL
LIN {X 0,Y 397.767,Z 709.334,A -85,B 0,C 180,E1 19514.398,E2 19514.398} C_VEL
LIN {X 0,Y 399.711,Z 699.492,A -85,B 0,C 180,E1 19511.931,E2 19511.931} C_VEL
LIN {X 0,Y 401.973,Z 688.118,A -85,B 0,C 180,E1 19509.621,E2 19509.621} C_VEL
LIN {X 0,Y 404.292,Z 676.096,A -85,B 0,C 180,E1 19507.614,E2 19507.614} C_VEL
LIN {X 0,Y 406.707,Z 662.704,A -85,B 0,C 180,E1 19505.761,E2 19505.761} C_VEL
LIN {X 0,Y 409.156,Z 647.802,A -85,B 0,C 180,E1 19504.065,E2 19504.065} C_VEL
LIN {X 0,Y 411.335,Z 632.67,A -85,B 0,C 180,E1 19502.652,E2 19502.652} C_VEL
LIN {X 0,Y 413.382,Z 615.861,A -85,B 0,C 180,E1 19501.387,E2 19501.387} C_VEL
LIN {X 0,Y 415.07,Z 597.887,A -85,B 0,C 180,E1 19500.329,E2 19500.329} C_VEL
LIN {X 0,Y 416.304,Z 579.433,A -85,B 0,C 180,E1 19499.522,E2 19499.522} C_VEL
LIN {X 0,Y 417.013,Z 560.547,A -85,B 0,C 180,E1 19498.955,E2 19498.955} C_VEL
LIN {X 0,Y 420.97,Z 370.964,A -85,B 0,C 180,E1 19495.716,E2 19495.716} C_VEL
LIN {X 0,Y 408.892,Z 349.416,A -85,B 0,C 180,E1 19493.948,E2 19493.948} C_VEL
LIN {X 0,Y 406.12,Z 344.736,A -85,B 0,C 180,E1 19493.498,E2 19493.498} C_VEL
LIN {X 0,Y 400.354,Z 329.96,A -85,B 0,C 180,E1 19490.734,E2 19490.734} C_VEL
LIN {X 0,Y 394.968,Z 317.07,A -85,B 0,C 180,E1 19488.064,E2 19488.064} C_VEL
LIN {X 0,Y 393.56,Z 313.603,A -85,B 0,C 180,E1 19487.242,E2 19487.242} C_VEL
LIN {X 0,Y 393.548,Z 313.459,A -85,B 0,C 180,E1 19483.513,E2 19483.513} C_VEL
LIN {X 0,Y 393.558,Z 313.465,A -85,B 0,C 180,E1 19479.62,E2 19479.62} C_VEL
LIN {X 0,Y 393.554,Z 313.463,A -85,B 0,C 180,E1 19475.614,E2 19475.614} C_VEL
LIN {X 0,Y 393.552,Z 313.464,A -85,B 0,C 180,E1 19471.559,E2 19471.559} C_VEL
LIN {X 0,Y 393.559,Z 313.459,A -85,B 0,C 180,E1 19467.706,E2 19467.706} C_VEL
LIN {X 0,Y 393.556,Z 313.446,A -85,B 0,C 180,E1 19463.667,E2 19463.667} C_VEL
LIN {X 0,Y 393.55,Z 313.44,A -85,B 0,C 180,E1 19459.749,E2 19459.749} C_VEL
LIN {X 0,Y 393.547,Z 313.451,A -85,B 0,C 180,E1 19455.775,E2 19455.775} C_VEL
LIN {X 0,Y 393.531,Z 313.462,A -85,B 0,C 180,E1 19451.877,E2 19451.877} C_VEL
LIN {X 0,Y 393.522,Z 313.442,A -85,B 0,C 180,E1 19447.886,E2 19447.886} C_VEL
LIN {X 0,Y 393.503,Z 313.452,A -85,B 0,C 180,E1 19444.08,E2 19444.08} C_VEL
LIN {X 0,Y 393.488,Z 313.468,A -85,B 0,C 180,E1 19440.291,E2 19440.291} C_VEL
LIN {X 0,Y 393.488,Z 313.45,A -85,B 0,C 180,E1 19436.358,E2 19436.358} C_VEL
LIN {X 0,Y 393.492,Z 313.448,A -85,B 0,C 180,E1 19432.408,E2 19432.408} C_VEL
LIN {X 0,Y 393.501,Z 313.467,A -85,B 0,C 180,E1 19428.42,E2 19428.42} C_VEL
LIN {X 0,Y 393.504,Z 313.467,A -85,B 0,C 180,E1 19424.36,E2 19424.36} C_VEL
LIN {X 0,Y 393.509,Z 313.457,A -85,B 0,C 180,E1 19420.404,E2 19420.404} C_VEL
LIN {X 0,Y 393.516,Z 313.45,A -85,B 0,C 180,E1 19416.49,E2 19416.49} C_VEL
LIN {X 0,Y 393.525,Z 313.449,A -85,B 0,C 180,E1 19412.621,E2 19412.621} C_VEL
LIN {X 0,Y 393.542,Z 313.449,A -85,B 0,C 180,E1 19408.782,E2 19408.782} C_VEL
LIN {X 0,Y 393.549,Z 313.409,A -85,B 0,C 180,E1 19404.891,E2 19404.891} C_VEL
LIN {X 0,Y 393.602,Z 313.683,A -85,B 0,C 180,E1 19401.138,E2 19401.138} C_VEL
LIN {X 0,Y 394.75,Z 316.793,A -85,B 0,C 180,E1 19400.524,E2 19400.524} C_VEL
LIN {X 0,Y 395.956,Z 318.911,A -85,B 0,C 180,E1 19400.104,E2 19400.104} C_VEL
LIN {X 0,Y 401.799,Z 330.761,A -85,B 0,C 180,E1 19397.98,E2 19397.98} C_VEL
LIN {X 0,Y 409.797,Z 348.447,A -85,B 0,C 180,E1 19395.161,E2 19395.161} C_VEL
LIN {X 0,Y 417.495,Z 367.578,A -85,B 0,C 180,E1 19392.471,E2 19392.471} C_VEL
LIN {X 0,Y 419.039,Z 372.186,A -85,B 0,C 180,E1 19391.888,E2 19391.888} C_VEL
LIN {X 0,Y 417.954,Z 382.538,A -85,B 0,C 180,E1 19391.074,E2 19391.074} C_VEL
LIN {X 0,Y 421.871,Z 422.728,A -85,B 0,C 180,E1 19389.787,E2 19389.787} C_VEL
LIN {X 0,Y 415.256,Z 635.275,A -85,B 0,C 180,E1 19385.721,E2 19385.721} C_VEL
LIN {X 0,Y 413.844,Z 656.322,A -85,B 0,C 180,E1 19385.123,E2 19385.123} C_VEL
LIN {X 0,Y 411.921,Z 676.513,A -85,B 0,C 180,E1 19384.314,E2 19384.314} C_VEL
LIN {X 0,Y 409.615,Z 696.882,A -85,B 0,C 180,E1 19383.229,E2 19383.229} C_VEL
LIN {X 0,Y 407.252,Z 715.888,A -85,B 0,C 180,E1 19381.942,E2 19381.942} C_VEL
LIN {X 0,Y 404.765,Z 734.249,A -85,B 0,C 180,E1 19380.423,E2 19380.423} C_VEL
LIN {X 0,Y 402.21,Z 752.538,A -85,B 0,C 180,E1 19378.589,E2 19378.589} C_VEL
LIN {X 0,Y 399.787,Z 769.779,A -85,B 0,C 180,E1 19376.514,E2 19376.514} C_VEL
LIN {X 0,Y 397.601,Z 785.904,A -85,B 0,C 180,E1 19374.198,E2 19374.198} C_VEL
LIN {X 0,Y 395.835,Z 799.983,A -85,B 0,C 180,E1 19371.796,E2 19371.796} C_VEL
LIN {X 0,Y 394.463,Z 812.649,A -85,B 0,C 180,E1 19369.239,E2 19369.239} C_VEL
LIN {X 0,Y 393.476,Z 823.859,A -85,B 0,C 180,E1 19366.535,E2 19366.535} C_VEL
LIN {X 0,Y 392.863,Z 833.534,A -85,B 0,C 180,E1 19363.691,E2 19363.691} C_VEL
LIN {X 0,Y 392.593,Z 841.224,A -85,B 0,C 180,E1 19360.863,E2 19360.863} C_VEL
LIN {X 0,Y 392.532,Z 847.083,A -85,B 0,C 180,E1 19358.053,E2 19358.053} C_VEL
LIN {X 0,Y 392.606,Z 851.096,A -85,B 0,C 180,E1 19355.26,E2 19355.26} C_VEL
LIN {X 0,Y 392.687,Z 853.424,A -85,B 0,C 180,E1 19352.481,E2 19352.481} C_VEL
LIN {X 0,Y 392.717,Z 854.138,A -85,B 0,C 180,E1 19349.854,E2 19349.854} C_VEL
LIN {X 0,Y 392.683,Z 853.267,A -85,B 0,C 180,E1 19347.227,E2 19347.227} C_VEL
LIN {X 0,Y 392.601,Z 850.733,A -85,B 0,C 180,E1 19344.447,E2 19344.447} C_VEL
LIN {X 0,Y 392.534,Z 846.526,A -85,B 0,C 180,E1 19341.652,E2 19341.652} C_VEL
LIN {X 0,Y 392.597,Z 840.885,A -85,B 0,C 180,E1 19338.989,E2 19338.989} C_VEL
LIN {X 0,Y 392.864,Z 833.534,A -85,B 0,C 180,E1 19336.309,E2 19336.309} C_VEL
LIN {X 0,Y 393.477,Z 823.854,A -85,B 0,C 180,E1 19333.465,E2 19333.465} C_VEL
LIN {X 0,Y 394.464,Z 812.641,A -85,B 0,C 180,E1 19330.761,E2 19330.761} C_VEL
LIN {X 0,Y 395.833,Z 799.971,A -85,B 0,C 180,E1 19328.204,E2 19328.204} C_VEL
LIN {X 0,Y 397.6,Z 785.884,A -85,B 0,C 180,E1 19325.802,E2 19325.802} C_VEL
LIN {X 0,Y 399.785,Z 769.75,A -85,B 0,C 180,E1 19323.486,E2 19323.486} C_VEL
LIN {X 0,Y 402.303,Z 751.833,A -85,B 0,C 180,E1 19321.337,E2 19321.337} C_VEL
LIN {X 0,Y 404.863,Z 733.507,A -85,B 0,C 180,E1 19319.511,E2 19319.511} C_VEL
LIN {X 0,Y 407.504,Z 713.952,A -85,B 0,C 180,E1 19317.914,E2 19317.914} C_VEL
LIN {X 0,Y 409.943,Z 694.091,A -85,B 0,C 180,E1 19316.607,E2 19316.607} C_VEL
LIN {X 0,Y 412.077,Z 674.905,A -85,B 0,C 180,E1 19315.617,E2 19315.617} C_VEL
LIN {X 0,Y 414.012,Z 653.942,A -85,B 0,C 180,E1 19314.802,E2 19314.802} C_VEL
LIN {X 0,Y 415.363,Z 632.112,A -85,B 0,C 180,E1 19314.215,E2 19314.215} C_VEL
LIN {X 0,Y 421.873,Z 421.052,A -85,B 0,C 180,E1 19310.186,E2 19310.186} C_VEL
LIN {X 0,Y 417.909,Z 381.477,A -85,B 0,C 180,E1 19308.879,E2 19308.879} C_VEL
LIN {X 0,Y 419.038,Z 371.813,A -85,B 0,C 180,E1 19308.081,E2 19308.081} C_VEL
LIN {X 0,Y 411.753,Z 353.239,A -85,B 0,C 180,E1 19305.554,E2 19305.554} C_VEL
LIN {X 0,Y 404.51,Z 336.713,A -85,B 0,C 180,E1 19303.016,E2 19303.016} C_VEL
LIN {X 0,Y 397.474,Z 321.825,A -85,B 0,C 180,E1 19300.466,E2 19300.466} C_VEL
LIN {X 0,Y 393.692,Z 314.172,A -85,B 0,C 180,E1 19299.033,E2 19299.033} C_VEL
LIN {X 0,Y 393.562,Z 313.469,A -85,B 0,C 180,E1 19298.68,E2 19298.68} C_VEL
LIN {X 0,Y 393.552,Z 313.417,A -85,B 0,C 180,E1 19294.687,E2 19294.687} C_VEL
LIN {X 0,Y 393.565,Z 313.448,A -85,B 0,C 180,E1 19290.706,E2 19290.706} C_VEL
LIN {X 0,Y 393.558,Z 313.448,A -85,B 0,C 180,E1 19286.723,E2 19286.723} C_VEL
LIN {X 0,Y 393.565,Z 313.444,A -85,B 0,C 180,E1 19282.715,E2 19282.715} C_VEL
LIN {X 0,Y 393.55,Z 313.443,A -85,B 0,C 180,E1 19278.67,E2 19278.67} C_VEL
LIN {X 0,Y 393.554,Z 313.448,A -85,B 0,C 180,E1 19274.717,E2 19274.717} C_VEL
LIN {X 0,Y 393.541,Z 313.466,A -85,B 0,C 180,E1 19270.688,E2 19270.688} C_VEL
LIN {X 0,Y 393.548,Z 313.454,A -85,B 0,C 180,E1 19266.608,E2 19266.608} C_VEL
LIN {X 0,Y 393.531,Z 313.44,A -85,B 0,C 180,E1 19262.621,E2 19262.621} C_VEL
LIN {X 0,Y 393.522,Z 313.456,A -85,B 0,C 180,E1 19258.689,E2 19258.689} C_VEL
LIN {X 0,Y 393.515,Z 313.464,A -85,B 0,C 180,E1 19254.751,E2 19254.751} C_VEL
LIN {X 0,Y 393.501,Z 313.442,A -85,B 0,C 180,E1 19250.936,E2 19250.936} C_VEL
LIN {X 0,Y 393.499,Z 313.457,A -85,B 0,C 180,E1 19247.079,E2 19247.079} C_VEL
LIN {X 0,Y 393.502,Z 313.467,A -85,B 0,C 180,E1 19243.162,E2 19243.162} C_VEL
LIN {X 0,Y 393.505,Z 313.455,A -85,B 0,C 180,E1 19239.162,E2 19239.162} C_VEL
LIN {X 0,Y 393.507,Z 313.444,A -85,B 0,C 180,E1 19235.213,E2 19235.213} C_VEL
LIN {X 0,Y 393.513,Z 313.453,A -85,B 0,C 180,E1 19231.231,E2 19231.231} C_VEL
LIN {X 0,Y 393.518,Z 313.46,A -85,B 0,C 180,E1 19227.235,E2 19227.235} C_VEL
LIN {X 0,Y 393.524,Z 313.464,A -85,B 0,C 180,E1 19223.338,E2 19223.338} C_VEL
LIN {X 0,Y 393.535,Z 313.458,A -85,B 0,C 180,E1 19219.426,E2 19219.426} C_VEL
LIN {X 0,Y 393.538,Z 313.431,A -85,B 0,C 180,E1 19215.474,E2 19215.474} C_VEL
LIN {X 0,Y 393.567,Z 313.66,A -85,B 0,C 180,E1 19212.613,E2 19212.613} C_VEL
LIN {X 0,Y 398.812,Z 326.272,A -85,B 0,C 180,E1 19209.899,E2 19209.899} C_VEL
LIN {X 0,Y 404.332,Z 340.049,A -85,B 0,C 180,E1 19207.225,E2 19207.225} C_VEL
LIN {X 0,Y 406.421,Z 345.401,A -85,B 0,C 180,E1 19206.322,E2 19206.322} C_VEL
LIN {X 0,Y 417.747,Z 365.108,A -85,B 0,C 180,E1 19204.638,E2 19204.638} C_VEL
LIN {X 0,Y 421.06,Z 371.655,A -85,B 0,C 180,E1 19204.156,E2 19204.156} C_VEL
LIN {X 0,Y 416.97,Z 560.855,A -85,B 0,C 180,E1 19200.941,E2 19200.941} C_VEL
LIN {X 0,Y 416.238,Z 580.043,A -85,B 0,C 180,E1 19200.359,E2 19200.359} C_VEL
LIN {X 0,Y 414.951,Z 598.933,A -85,B 0,C 180,E1 19199.521,E2 19199.521} C_VEL
LIN {X 0,Y 413.27,Z 616.635,A -85,B 0,C 180,E1 19198.464,E2 19198.464} C_VEL
LIN {X 0,Y 411.226,Z 633.289,A -85,B 0,C 180,E1 19197.2,E2 19197.2} C_VEL
LIN {X 0,Y 408.847,Z 649.658,A -85,B 0,C 180,E1 19195.649,E2 19195.649} C_VEL
LIN {X 0,Y 406.337,Z 664.754,A -85,B 0,C 180,E1 19193.884,E2 19193.884} C_VEL
LIN {X 0,Y 403.855,Z 678.401,A -85,B 0,C 180,E1 19191.937,E2 19191.937} C_VEL
LIN {X 0,Y 401.943,Z 683.676,A -85,B 0,C 180,E1 19191.153,E2 19191.153} C_VEL
LIN {X 0,Y 393.99,Z 696.367,A -85,B 0,C 180,E1 19189.222,E2 19189.222} C_VEL
LIN {X 0,Y 392.177,Z 700.714,A -85,B 0,C 180,E1 19188.337,E2 19188.337} C_VEL
LIN {X 0,Y 390.193,Z 710.225,A -85,B 0,C 180,E1 19185.913,E2 19185.913} C_VEL
LIN {X 0,Y 388.465,Z 718.608,A -85,B 0,C 180,E1 19183.242,E2 19183.242} C_VEL
LIN {X 0,Y 387.22,Z 725.118,A -85,B 0,C 180,E1 19180.564,E2 19180.564} C_VEL
LIN {X 0,Y 386.334,Z 730.204,A -85,B 0,C 180,E1 19177.734,E2 19177.734} C_VEL
LIN {X 0,Y 385.788,Z 733.618,A -85,B 0,C 180,E1 19174.906,E2 19174.906} C_VEL
LIN {X 0,Y 385.519,Z 735.537,A -85,B 0,C 180,E1 19171.932,E2 19171.932} C_VEL
LIN {X 0,Y 385.481,Z 735.811,A -85,B 0,C 180,E1 19168.96,E2 19168.96} C_VEL
LIN {X 0,Y 385.669,Z 734.451,A -85,B 0,C 180,E1 19165.986,E2 19165.986} C_VEL
LIN {X 0,Y 386.108,Z 731.587,A -85,B 0,C 180,E1 19163.159,E2 19163.159} C_VEL
LIN {X 0,Y 386.879,Z 727.097,A -85,B 0,C 180,E1 19160.329,E2 19160.329} C_VEL
LIN {X 0,Y 388.037,Z 720.843,A -85,B 0,C 180,E1 19157.5,E2 19157.5} C_VEL
LIN {X 0,Y 389.611,Z 713.082,A -85,B 0,C 180,E1 19154.826,E2 19154.826} C_VEL
LIN {X 0,Y 391.536,Z 703.858,A -85,B 0,C 180,E1 19152.309,E2 19152.309} C_VEL
LIN {X 0,Y 393.775,Z 693.191,A -85,B 0,C 180,E1 19149.954,E2 19149.954} C_VEL
LIN {X 0,Y 396.276,Z 681.051,A -85,B 0,C 180,E1 19147.762,E2 19147.762} C_VEL
LIN {X 0,Y 398.813,Z 667.874,A -85,B 0,C 180,E1 19145.802,E2 19145.802} C_VEL
LIN {X 0,Y 401.423,Z 653.145,A -85,B 0,C 180,E1 19144,E2 19144} C_VEL
LIN {X 0,Y 403.781,Z 638.127,A -85,B 0,C 180,E1 19142.496,E2 19142.496} C_VEL
LIN {X 0,Y 406.017,Z 621.425,A -85,B 0,C 180,E1 19141.141,E2 19141.141} C_VEL
LIN {X 0,Y 407.797,Z 604.816,A -85,B 0,C 180,E1 19140.07,E2 19140.07} C_VEL
LIN {X 0,Y 409.272,Z 586.2,A -85,B 0,C 180,E1 19139.155,E2 19139.155} C_VEL
LIN {X 0,Y 410.213,Z 566.946,A -85,B 0,C 180,E1 19138.489,E2 19138.489} C_VEL
LIN {X 0,Y 410.706,Z 542.868,A -85,B 0,C 180,E1 19137.988,E2 19137.988} C_VEL
LIN {X 0,Y 414.637,Z 373.964,A -85,B 0,C 180,E1 19135.1,E2 19135.1} C_VEL
LIN {X 0,Y 403.294,Z 353.738,A -85,B 0,C 180,E1 19133.385,E2 19133.385} C_VEL
LIN {X 0,Y 398.148,Z 345.046,A -85,B 0,C 180,E1 19132.52,E2 19132.52} C_VEL
LIN {X 0,Y 391.902,Z 329.245,A -85,B 0,C 180,E1 19129.416,E2 19129.416} C_VEL
LIN {X 0,Y 387.041,Z 318.11,A -85,B 0,C 180,E1 19126.978,E2 19126.978} C_VEL
LIN {X 0,Y 385.647,Z 314.605,A -85,B 0,C 180,E1 19126.118,E2 19126.118} C_VEL
LIN {X 0,Y 385.622,Z 314.44,A -85,B 0,C 180,E1 19122.138,E2 19122.138} C_VEL
LIN {X 0,Y 385.621,Z 314.435,A -85,B 0,C 180,E1 19118.105,E2 19118.105} C_VEL
LIN {X 0,Y 385.615,Z 314.434,A -85,B 0,C 180,E1 19114.061,E2 19114.061} C_VEL
LIN {X 0,Y 385.617,Z 314.433,A -85,B 0,C 180,E1 19110.003,E2 19110.003} C_VEL
LIN {X 0,Y 385.599,Z 314.444,A -85,B 0,C 180,E1 19106.156,E2 19106.156} C_VEL
LIN {X 0,Y 385.588,Z 314.455,A -85,B 0,C 180,E1 19102.226,E2 19102.226} C_VEL
LIN {X 0,Y 385.578,Z 314.444,A -85,B 0,C 180,E1 19098.287,E2 19098.287} C_VEL
LIN {X 0,Y 385.566,Z 314.43,A -85,B 0,C 180,E1 19094.416,E2 19094.416} C_VEL
LIN {X 0,Y 385.563,Z 314.453,A -85,B 0,C 180,E1 19090.459,E2 19090.459} C_VEL
LIN {X 0,Y 385.555,Z 314.456,A -85,B 0,C 180,E1 19086.552,E2 19086.552} C_VEL
LIN {X 0,Y 385.548,Z 314.432,A -85,B 0,C 180,E1 19082.527,E2 19082.527} C_VEL
LIN {X 0,Y 385.547,Z 314.444,A -85,B 0,C 180,E1 19078.514,E2 19078.514} C_VEL
LIN {X 0,Y 385.554,Z 314.456,A -85,B 0,C 180,E1 19074.494,E2 19074.494} C_VEL
LIN {X 0,Y 385.558,Z 314.445,A -85,B 0,C 180,E1 19070.447,E2 19070.447} C_VEL
LIN {X 0,Y 385.561,Z 314.432,A -85,B 0,C 180,E1 19066.351,E2 19066.351} C_VEL
LIN {X 0,Y 385.566,Z 314.441,A -85,B 0,C 180,E1 19062.338,E2 19062.338} C_VEL
LIN {X 0,Y 385.572,Z 314.449,A -85,B 0,C 180,E1 19058.234,E2 19058.234} C_VEL
LIN {X 0,Y 385.579,Z 314.451,A -85,B 0,C 180,E1 19054.131,E2 19054.131} C_VEL
LIN {X 0,Y 385.58,Z 314.45,A -85,B 0,C 180,E1 19050.14,E2 19050.14} C_VEL
LIN {X 0,Y 385.581,Z 314.427,A -85,B 0,C 180,E1 19046.076,E2 19046.076} C_VEL
LIN {X 0,Y 385.606,Z 314.558,A -85,B 0,C 180,E1 19042.365,E2 19042.365} C_VEL
LIN {X 0,Y 386.069,Z 316.334,A -85,B 0,C 180,E1 19041.948,E2 19041.948} C_VEL
LIN {X 0,Y 387.999,Z 319.736,A -85,B 0,C 180,E1 19041.23,E2 19041.23} C_VEL
LIN {X 0,Y 394.474,Z 332.948,A -85,B 0,C 180,E1 19038.776,E2 19038.776} C_VEL
LIN {X 0,Y 402.152,Z 349.684,A -85,B 0,C 180,E1 19035.98,E2 19035.98} C_VEL
LIN {X 0,Y 409.948,Z 368.876,A -85,B 0,C 180,E1 19033.176,E2 19033.176} C_VEL
LIN {X 0,Y 412.124,Z 375.317,A -85,B 0,C 180,E1 19032.316,E2 19032.316} C_VEL
LIN {X 0,Y 411.447,Z 382.221,A -85,B 0,C 180,E1 19031.784,E2 19031.784} C_VEL
LIN {X 0,Y 415.419,Z 423.705,A -85,B 0,C 180,E1 19030.425,E2 19030.425} C_VEL
LIN {X 0,Y 408.519,Z 634.944,A -85,B 0,C 180,E1 19026.328,E2 19026.328} C_VEL
LIN {X 0,Y 407.039,Z 655.856,A -85,B 0,C 180,E1 19025.721,E2 19025.721} C_VEL
LIN {X 0,Y 405.023,Z 676.041,A -85,B 0,C 180,E1 19024.896,E2 19024.896} C_VEL
LIN {X 0,Y 402.603,Z 696.28,A -85,B 0,C 180,E1 19023.799,E2 19023.799} C_VEL
LIN {X 0,Y 399.99,Z 716.125,A -85,B 0,C 180,E1 19022.423,E2 19022.423} C_VEL
LIN {X 0,Y 397.388,Z 734.247,A -85,B 0,C 180,E1 19020.881,E2 19020.881} C_VEL
LIN {X 0,Y 394.81,Z 751.702,A -85,B 0,C 180,E1 19019.093,E2 19019.093} C_VEL
LIN {X 0,Y 392.246,Z 768.898,A -85,B 0,C 180,E1 19016.982,E2 19016.982} C_VEL
LIN {X 0,Y 389.928,Z 784.982,A -85,B 0,C 180,E1 19014.625,E2 19014.625} C_VEL
LIN {X 0,Y 388.003,Z 799.438,A -85,B 0,C 180,E1 19012.1,E2 19012.1} C_VEL
LIN {X 0,Y 386.562,Z 811.997,A -85,B 0,C 180,E1 19009.491,E2 19009.491} C_VEL
LIN {X 0,Y 385.527,Z 823.11,A -85,B 0,C 180,E1 19006.73,E2 19006.73} C_VEL
LIN {X 0,Y 384.897,Z 832.698,A -85,B 0,C 180,E1 19003.827,E2 19003.827} C_VEL
LIN {X 0,Y 384.626,Z 840.306,A -85,B 0,C 180,E1 19000.939,E2 19000.939} C_VEL
LIN {X 0,Y 384.583,Z 845.847,A -85,B 0,C 180,E1 18998.221,E2 18998.221} C_VEL
LIN {X 0,Y 384.675,Z 849.795,A -85,B 0,C 180,E1 18995.437,E2 18995.437} C_VEL
LIN {X 0,Y 384.771,Z 852.141,A -85,B 0,C 180,E1 18992.681,E2 18992.681} C_VEL
LIN {X 0,Y 384.812,Z 852.954,A -85,B 0,C 180,E1 18990,E2 18990} C_VEL
LIN {X 0,Y 384.772,Z 852.14,A -85,B 0,C 180,E1 18987.319,E2 18987.319} C_VEL
LIN {X 0,Y 384.673,Z 849.694,A -85,B 0,C 180,E1 18984.481,E2 18984.481} C_VEL
LIN {X 0,Y 384.583,Z 845.846,A -85,B 0,C 180,E1 18981.779,E2 18981.779} C_VEL
LIN {X 0,Y 384.632,Z 839.966,A -85,B 0,C 180,E1 18978.909,E2 18978.909} C_VEL
LIN {X 0,Y 384.897,Z 832.697,A -85,B 0,C 180,E1 18976.173,E2 18976.173} C_VEL
LIN {X 0,Y 385.527,Z 823.103,A -85,B 0,C 180,E1 18973.27,E2 18973.27} C_VEL
LIN {X 0,Y 386.562,Z 811.985,A -85,B 0,C 180,E1 18970.509,E2 18970.509} C_VEL
LIN {X 0,Y 388.003,Z 799.422,A -85,B 0,C 180,E1 18967.9,E2 18967.9} C_VEL
LIN {X 0,Y 389.927,Z 784.958,A -85,B 0,C 180,E1 18965.375,E2 18965.375} C_VEL
LIN {X 0,Y 392.244,Z 768.864,A -85,B 0,C 180,E1 18963.017,E2 18963.017} C_VEL
LIN {X 0,Y 394.897,Z 751.073,A -85,B 0,C 180,E1 18960.839,E2 18960.839} C_VEL
LIN {X 0,Y 397.624,Z 732.652,A -85,B 0,C 180,E1 18958.971,E2 18958.971} C_VEL
LIN {X 0,Y 400.293,Z 713.881,A -85,B 0,C 180,E1 18957.407,E2 18957.407} C_VEL
LIN {X 0,Y 402.784,Z 694.725,A -85,B 0,C 180,E1 18956.111,E2 18956.111} C_VEL
LIN {X 0,Y 405.099,Z 675.163,A -85,B 0,C 180,E1 18955.068,E2 18955.068} C_VEL
LIN {X 0,Y 407.181,Z 653.862,A -85,B 0,C 180,E1 18954.217,E2 18954.217} C_VEL
LIN {X 0,Y 408.624,Z 631.863,A -85,B 0,C 180,E1 18953.61,E2 18953.61} C_VEL
LIN {X 0,Y 415.42,Z 422.205,A -85,B 0,C 180,E1 18949.553,E2 18949.553} C_VEL
LIN {X 0,Y 411.396,Z 380.893,A -85,B 0,C 180,E1 18948.154,E2 18948.154} C_VEL
LIN {X 0,Y 412.119,Z 374.753,A -85,B 0,C 180,E1 18947.625,E2 18947.625} C_VEL
LIN {X 0,Y 404.692,Z 355.738,A -85,B 0,C 180,E1 18944.959,E2 18944.959} C_VEL
LIN {X 0,Y 397.175,Z 338.608,A -85,B 0,C 180,E1 18942.233,E2 18942.233} C_VEL
LIN {X 0,Y 389.71,Z 323.102,A -85,B 0,C 180,E1 18939.445,E2 18939.445} C_VEL
LIN {X 0,Y 387.178,Z 318.289,A -85,B 0,C 180,E1 18938.489,E2 18938.489} C_VEL
LIN {X 0,Y 385.625,Z 314.681,A -85,B 0,C 180,E1 18937.727,E2 18937.727} C_VEL
LIN {X 0,Y 385.601,Z 314.41,A -85,B 0,C 180,E1 18934.458,E2 18934.458} C_VEL
LIN {X 0,Y 385.614,Z 314.439,A -85,B 0,C 180,E1 18930.544,E2 18930.544} C_VEL
LIN {X 0,Y 385.611,Z 314.438,A -85,B 0,C 180,E1 18926.552,E2 18926.552} C_VEL
LIN {X 0,Y 385.614,Z 314.434,A -85,B 0,C 180,E1 18922.566,E2 18922.566} C_VEL
LIN {X 0,Y 385.609,Z 314.431,A -85,B 0,C 180,E1 18918.598,E2 18918.598} C_VEL
LIN {X 0,Y 385.615,Z 314.434,A -85,B 0,C 180,E1 18914.567,E2 18914.567} C_VEL
LIN {X 0,Y 385.6,Z 314.451,A -85,B 0,C 180,E1 18910.457,E2 18910.457} C_VEL
LIN {X 0,Y 385.6,Z 314.446,A -85,B 0,C 180,E1 18906.401,E2 18906.401} C_VEL
LIN {X 0,Y 385.589,Z 314.429,A -85,B 0,C 180,E1 18902.378,E2 18902.378} C_VEL
LIN {X 0,Y 385.593,Z 314.44,A -85,B 0,C 180,E1 18898.514,E2 18898.514} C_VEL
LIN {X 0,Y 385.594,Z 314.456,A -85,B 0,C 180,E1 18894.345,E2 18894.345} C_VEL
LIN {X 0,Y 385.592,Z 314.431,A -85,B 0,C 180,E1 18890.447,E2 18890.447} C_VEL
LIN {X 0,Y 385.607,Z 314.428,A -85,B 0,C 180,E1 18886.352,E2 18886.352} C_VEL
LIN {X 0,Y 385.607,Z 314.448,A -85,B 0,C 180,E1 18882.339,E2 18882.339} C_VEL
LIN {X 0,Y 385.621,Z 314.448,A -85,B 0,C 180,E1 18878.236,E2 18878.236} C_VEL
LIN {X 0,Y 385.611,Z 314.436,A -85,B 0,C 180,E1 18874.121,E2 18874.121} C_VEL
LIN {X 0,Y 385.629,Z 314.431,A -85,B 0,C 180,E1 18870.144,E2 18870.144} C_VEL
LIN {X 0,Y 385.618,Z 314.434,A -85,B 0,C 180,E1 18866.067,E2 18866.067} C_VEL
LIN {X 0,Y 385.625,Z 314.435,A -85,B 0,C 180,E1 18862.017,E2 18862.017} C_VEL
LIN {X 0,Y 385.624,Z 314.438,A -85,B 0,C 180,E1 18858.013,E2 18858.013} C_VEL
LIN {X 0,Y 385.626,Z 314.47,A -85,B 0,C 180,E1 18853.879,E2 18853.879} C_VEL
LIN {X 0,Y 385.859,Z 315.653,A -85,B 0,C 180,E1 18853.485,E2 18853.485} C_VEL
LIN {X 0,Y 389.443,Z 323.771,A -85,B 0,C 180,E1 18851.658,E2 18851.658} C_VEL
LIN {X 0,Y 394.691,Z 336.105,A -85,B 0,C 180,E1 18849.075,E2 18849.075} C_VEL
LIN {X 0,Y 398.547,Z 345.9,A -85,B 0,C 180,E1 18847.259,E2 18847.259} C_VEL
LIN {X 0,Y 410.134,Z 365.728,A -85,B 0,C 180,E1 18845.461,E2 18845.461} C_VEL
LIN {X 0,Y 414.661,Z 374.464,A -85,B 0,C 180,E1 18844.781,E2 18844.781} C_VEL
LIN {X 0,Y 410.35,Z 561.559,A -85,B 0,C 180,E1 18841.555,E2 18841.555} C_VEL
LIN {X 0,Y 409.587,Z 580.645,A -85,B 0,C 180,E1 18840.971,E2 18840.971} C_VEL
LIN {X 0,Y 408.262,Z 599.362,A -85,B 0,C 180,E1 18840.135,E2 18840.135} C_VEL
LIN {X 0,Y 406.502,Z 617.193,A -85,B 0,C 180,E1 18839.063,E2 18839.063} C_VEL
LIN {X 0,Y 404.361,Z 633.932,A -85,B 0,C 180,E1 18837.781,E2 18837.781} C_VEL
LIN {X 0,Y 401.982,Z 649.691,A -85,B 0,C 180,E1 18836.278,E2 18836.278} C_VEL
LIN {X 0,Y 399.332,Z 665.051,A -85,B 0,C 180,E1 18834.48,E2 18834.48} C_VEL
LIN {X 0,Y 396.734,Z 678.706,A -85,B 0,C 180,E1 18832.524,E2 18832.524} C_VEL
LIN {X 0,Y 394.177,Z 691.263,A -85,B 0,C 180,E1 18830.335,E2 18830.335} C_VEL
LIN {X 0,Y 392.177,Z 700.714,A -85,B 0,C 180,E1 18828.337,E2 18828.337} C_VEL
LIN {X 0,Y 390.401,Z 704.945,A -85,B 0,C 180,E1 18827.419,E2 18827.419} C_VEL
LIN {X 0,Y 383.096,Z 714.504,A -85,B 0,C 180,E1 18825.235,E2 18825.235} C_VEL
LIN {X 0,Y 381.201,Z 717.867,A -85,B 0,C 180,E1 18824.223,E2 18824.223} C_VEL
LIN {X 0,Y 381.081,Z 718.294,A -85,B 0,C 180,E1 18824.07,E2 18824.07} C_VEL
LIN {X 0,Y 379.62,Z 725.372,A -85,B 0,C 180,E1 18821.239,E2 18821.239} C_VEL
LIN {X 0,Y 378.609,Z 730.728,A -85,B 0,C 180,E1 18818.351,E2 18818.351} C_VEL
LIN {X 0,Y 377.947,Z 734.538,A -85,B 0,C 180,E1 18815.313,E2 18815.313} C_VEL
LIN {X 0,Y 377.628,Z 736.618,A -85,B 0,C 180,E1 18812.276,E2 18812.276} C_VEL
LIN {X 0,Y 377.569,Z 737.051,A -85,B 0,C 180,E1 18809.241,E2 18809.241} C_VEL
LIN {X 0,Y 377.738,Z 735.857,A -85,B 0,C 180,E1 18806.206,E2 18806.206} C_VEL
LIN {X 0,Y 378.21,Z 732.98,A -85,B 0,C 180,E1 18803.168,E2 18803.168} C_VEL
LIN {X 0,Y 379.011,Z 728.584,A -85,B 0,C 180,E1 18800.28,E2 18800.28} C_VEL
LIN {X 0,Y 380.217,Z 722.434,A -85,B 0,C 180,E1 18797.393,E2 18797.393} C_VEL
LIN {X 0,Y 381.855,Z 714.787,A -85,B 0,C 180,E1 18794.666,E2 18794.666} C_VEL
LIN {X 0,Y 383.859,Z 705.693,A -85,B 0,C 180,E1 18792.1,E2 18792.1} C_VEL
LIN {X 0,Y 386.186,Z 695.176,A -85,B 0,C 180,E1 18789.701,E2 18789.701} C_VEL
LIN {X 0,Y 388.781,Z 683.214,A -85,B 0,C 180,E1 18787.469,E2 18787.469} C_VEL
LIN {X 0,Y 391.557,Z 669.548,A -85,B 0,C 180,E1 18785.377,E2 18785.377} C_VEL
LIN {X 0,Y 394.32,Z 654.709,A -85,B 0,C 180,E1 18783.52,E2 18783.52} C_VEL
LIN {X 0,Y 396.938,Z 638.786,A -85,B 0,C 180,E1 18781.899,E2 18781.899} C_VEL
LIN {X 0,Y 399.22,Z 622.45,A -85,B 0,C 180,E1 18780.558,E2 18780.558} C_VEL
LIN {X 0,Y 401.139,Z 605.268,A -85,B 0,C 180,E1 18779.438,E2 18779.438} C_VEL
LIN {X 0,Y 402.681,Z 586.474,A -85,B 0,C 180,E1 18778.51,E2 18778.51} C_VEL
LIN {X 0,Y 403.641,Z 567.558,A -85,B 0,C 180,E1 18777.853,E2 18777.853} C_VEL
LIN {X 0,Y 404.166,Z 543.341,A -85,B 0,C 180,E1 18777.344,E2 18777.344} C_VEL
LIN {X 0,Y 408.292,Z 376.865,A -85,B 0,C 180,E1 18774.457,E2 18774.457} C_VEL
LIN {X 0,Y 397.395,Z 357.5,A -85,B 0,C 180,E1 18772.751,E2 18772.751} C_VEL
LIN {X 0,Y 390.285,Z 345.742,A -85,B 0,C 180,E1 18771.54,E2 18771.54} C_VEL
LIN {X 0,Y 384.365,Z 330.944,A -85,B 0,C 180,E1 18768.52,E2 18768.52} C_VEL
LIN {X 0,Y 379.18,Z 319.159,A -85,B 0,C 180,E1 18765.827,E2 18765.827} C_VEL
LIN {X 0,Y 377.685,Z 315.625,A -85,B 0,C 180,E1 18764.919,E2 18764.919} C_VEL
LIN {X 0,Y 377.652,Z 315.43,A -85,B 0,C 180,E1 18761.015,E2 18761.015} C_VEL
LIN {X 0,Y 377.648,Z 315.433,A -85,B 0,C 180,E1 18756.913,E2 18756.913} C_VEL
LIN {X 0,Y 377.644,Z 315.432,A -85,B 0,C 180,E1 18752.872,E2 18752.872} C_VEL
LIN {X 0,Y 377.64,Z 315.427,A -85,B 0,C 180,E1 18748.795,E2 18748.795} C_VEL
LIN {X 0,Y 377.636,Z 315.42,A -85,B 0,C 180,E1 18744.73,E2 18744.73} C_VEL
LIN {X 0,Y 377.634,Z 315.428,A -85,B 0,C 180,E1 18740.619,E2 18740.619} C_VEL
LIN {X 0,Y 377.63,Z 315.444,A -85,B 0,C 180,E1 18736.575,E2 18736.575} C_VEL
LIN {X 0,Y 377.623,Z 315.438,A -85,B 0,C 180,E1 18732.54,E2 18732.54} C_VEL
LIN {X 0,Y 377.616,Z 315.417,A -85,B 0,C 180,E1 18728.527,E2 18728.527} C_VEL
LIN {X 0,Y 377.614,Z 315.439,A -85,B 0,C 180,E1 18724.556,E2 18724.556} C_VEL
LIN {X 0,Y 377.61,Z 315.445,A -85,B 0,C 180,E1 18720.455,E2 18720.455} C_VEL
LIN {X 0,Y 377.611,Z 315.425,A -85,B 0,C 180,E1 18716.357,E2 18716.357} C_VEL
LIN {X 0,Y 377.615,Z 315.423,A -85,B 0,C 180,E1 18712.393,E2 18712.393} C_VEL
LIN {X 0,Y 377.623,Z 315.445,A -85,B 0,C 180,E1 18708.391,E2 18708.391} C_VEL
LIN {X 0,Y 377.627,Z 315.445,A -85,B 0,C 180,E1 18704.332,E2 18704.332} C_VEL
LIN {X 0,Y 377.632,Z 315.437,A -85,B 0,C 180,E1 18700.19,E2 18700.19} C_VEL
LIN {X 0,Y 377.636,Z 315.43,A -85,B 0,C 180,E1 18696.103,E2 18696.103} C_VEL
LIN {X 0,Y 377.641,Z 315.43,A -85,B 0,C 180,E1 18692.055,E2 18692.055} C_VEL
LIN {X 0,Y 377.646,Z 315.434,A -85,B 0,C 180,E1 18688.027,E2 18688.027} C_VEL
LIN {X 0,Y 377.641,Z 315.379,A -85,B 0,C 180,E1 18684.001,E2 18684.001} C_VEL
LIN {X 0,Y 377.755,Z 315.934,A -85,B 0,C 180,E1 18683.449,E2 18683.449} C_VEL
LIN {X 0,Y 379.388,Z 319.449,A -85,B 0,C 180,E1 18682.688,E2 18682.688} C_VEL
LIN {X 0,Y 384.547,Z 329.646,A -85,B 0,C 180,E1 18680.623,E2 18680.623} C_VEL
LIN {X 0,Y 391.456,Z 344.031,A -85,B 0,C 180,E1 18677.995,E2 18677.995} C_VEL
LIN {X 0,Y 398.852,Z 361.24,A -85,B 0,C 180,E1 18675.218,E2 18675.218} C_VEL
LIN {X 0,Y 405.282,Z 378.055,A -85,B 0,C 180,E1 18672.793,E2 18672.793} C_VEL
LIN {X 0,Y 404.997,Z 381.83,A -85,B 0,C 180,E1 18672.52,E2 18672.52} C_VEL
LIN {X 0,Y 409.019,Z 424.703,A -85,B 0,C 180,E1 18671.082,E2 18671.082} C_VEL
LIN {X 0,Y 401.833,Z 634.597,A -85,B 0,C 180,E1 18666.956,E2 18666.956} C_VEL
LIN {X 0,Y 400.258,Z 655.687,A -85,B 0,C 180,E1 18666.33,E2 18666.33} C_VEL
LIN {X 0,Y 398.177,Z 675.511,A -85,B 0,C 180,E1 18665.502,E2 18665.502} C_VEL
LIN {X 0,Y 395.638,Z 695.694,A -85,B 0,C 180,E1 18664.389,E2 18664.389} C_VEL
LIN {X 0,Y 392.895,Z 715.442,A -85,B 0,C 180,E1 18662.996,E2 18662.996} C_VEL
LIN {X 0,Y 390.04,Z 734.256,A -85,B 0,C 180,E1 18661.357,E2 18661.357} C_VEL
LIN {X 0,Y 387.334,Z 751.52,A -85,B 0,C 180,E1 18659.54,E2 18659.54} C_VEL
LIN {X 0,Y 384.645,Z 768.562,A -85,B 0,C 180,E1 18657.393,E2 18657.393} C_VEL
LIN {X 0,Y 382.278,Z 784.065,A -85,B 0,C 180,E1 18655.069,E2 18655.069} C_VEL
LIN {X 0,Y 380.185,Z 798.898,A -85,B 0,C 180,E1 18652.416,E2 18652.416} C_VEL
LIN {X 0,Y 378.593,Z 812.046,A -85,B 0,C 180,E1 18649.597,E2 18649.597} C_VEL
LIN {X 0,Y 377.535,Z 822.936,A -85,B 0,C 180,E1 18646.778,E2 18646.778} C_VEL
LIN {X 0,Y 376.93,Z 831.868,A -85,B 0,C 180,E1 18643.968,E2 18643.968} C_VEL
LIN {X 0,Y 376.66,Z 839.392,A -85,B 0,C 180,E1 18641.018,E2 18641.018} C_VEL
LIN {X 0,Y 376.635,Z 844.855,A -85,B 0,C 180,E1 18638.242,E2 18638.242} C_VEL
LIN {X 0,Y 376.743,Z 848.66,A -85,B 0,C 180,E1 18635.482,E2 18635.482} C_VEL
LIN {X 0,Y 376.858,Z 851.014,A -85,B 0,C 180,E1 18632.585,E2 18632.585} C_VEL
LIN {X 0,Y 376.898,Z 851.734,A -85,B 0,C 180,E1 18629.848,E2 18629.848} C_VEL
LIN {X 0,Y 376.848,Z 850.855,A -85,B 0,C 180,E1 18627.11,E2 18627.11} C_VEL
LIN {X 0,Y 376.723,Z 848.292,A -85,B 0,C 180,E1 18624.212,E2 18624.212} C_VEL
LIN {X 0,Y 376.629,Z 844.329,A -85,B 0,C 180,E1 18621.451,E2 18621.451} C_VEL
LIN {X 0,Y 376.679,Z 838.365,A -85,B 0,C 180,E1 18618.517,E2 18618.517} C_VEL
LIN {X 0,Y 377.01,Z 830.51,A -85,B 0,C 180,E1 18615.565,E2 18615.565} C_VEL
LIN {X 0,Y 377.68,Z 821.222,A -85,B 0,C 180,E1 18612.753,E2 18612.753} C_VEL
LIN {X 0,Y 378.829,Z 809.95,A -85,B 0,C 180,E1 18609.934,E2 18609.934} C_VEL
LIN {X 0,Y 380.405,Z 797.214,A -85,B 0,C 180,E1 18607.271,E2 18607.271} C_VEL
LIN {X 0,Y 382.417,Z 783.045,A -85,B 0,C 180,E1 18604.775,E2 18604.775} C_VEL
LIN {X 0,Y 384.818,Z 767.421,A -85,B 0,C 180,E1 18602.453,E2 18602.453} C_VEL
LIN {X 0,Y 387.539,Z 750.183,A -85,B 0,C 180,E1 18600.307,E2 18600.307} C_VEL
LIN {X 0,Y 390.414,Z 731.886,A -85,B 0,C 180,E1 18598.418,E2 18598.418} C_VEL
LIN {X 0,Y 393.164,Z 713.487,A -85,B 0,C 180,E1 18596.856,E2 18596.856} C_VEL
LIN {X 0,Y 395.788,Z 694.418,A -85,B 0,C 180,E1 18595.538,E2 18595.538} C_VEL
LIN {X 0,Y 398.245,Z 674.689,A -85,B 0,C 180,E1 18594.465,E2 18594.465} C_VEL
LIN {X 0,Y 400.389,Z 653.874,A -85,B 0,C 180,E1 18593.615,E2 18593.615} C_VEL
LIN {X 0,Y 401.888,Z 632.696,A -85,B 0,C 180,E1 18593.008,E2 18593.008} C_VEL
LIN {X 0,Y 409.017,Z 423.458,A -85,B 0,C 180,E1 18588.902,E2 18588.902} C_VEL
LIN {X 0,Y 404.926,Z 380.548,A -85,B 0,C 180,E1 18587.425,E2 18587.425} C_VEL
LIN {X 0,Y 405.115,Z 377.496,A -85,B 0,C 180,E1 18587.14,E2 18587.14} C_VEL
LIN {X 0,Y 398.239,Z 359.716,A -85,B 0,C 180,E1 18584.566,E2 18584.566} C_VEL
LIN {X 0,Y 391.007,Z 343.145,A -85,B 0,C 180,E1 18581.867,E2 18581.867} C_VEL
LIN {X 0,Y 384.173,Z 328.694,A -85,B 0,C 180,E1 18579.23,E2 18579.23} C_VEL
LIN {X 0,Y 379.333,Z 319.376,A -85,B 0,C 180,E1 18577.318,E2 18577.318} C_VEL
LIN {X 0,Y 377.714,Z 315.727,A -85,B 0,C 180,E1 18576.508,E2 18576.508} C_VEL
LIN {X 0,Y 377.672,Z 315.384,A -85,B 0,C 180,E1 18575.064,E2 18575.064} C_VEL
LIN {X 0,Y 377.674,Z 315.425,A -85,B 0,C 180,E1 18571.08,E2 18571.08} C_VEL
LIN {X 0,Y 377.666,Z 315.425,A -85,B 0,C 180,E1 18567.088,E2 18567.088} C_VEL
LIN {X 0,Y 377.66,Z 315.423,A -85,B 0,C 180,E1 18563.068,E2 18563.068} C_VEL
LIN {X 0,Y 377.653,Z 315.424,A -85,B 0,C 180,E1 18559.065,E2 18559.065} C_VEL
LIN {X 0,Y 377.649,Z 315.434,A -85,B 0,C 180,E1 18555.038,E2 18555.038} C_VEL
LIN {X 0,Y 377.645,Z 315.444,A -85,B 0,C 180,E1 18550.989,E2 18550.989} C_VEL
LIN {X 0,Y 377.637,Z 315.43,A -85,B 0,C 180,E1 18546.995,E2 18546.995} C_VEL
LIN {X 0,Y 377.626,Z 315.42,A -85,B 0,C 180,E1 18543.035,E2 18543.035} C_VEL
LIN {X 0,Y 377.621,Z 315.443,A -85,B 0,C 180,E1 18539.089,E2 18539.089} C_VEL
LIN {X 0,Y 377.616,Z 315.441,A -85,B 0,C 180,E1 18535.139,E2 18535.139} C_VEL
LIN {X 0,Y 377.614,Z 315.418,A -85,B 0,C 180,E1 18531.166,E2 18531.166} C_VEL
LIN {X 0,Y 377.621,Z 315.434,A -85,B 0,C 180,E1 18527.149,E2 18527.149} C_VEL
LIN {X 0,Y 377.625,Z 315.445,A -85,B 0,C 180,E1 18523.225,E2 18523.225} C_VEL
LIN {X 0,Y 377.628,Z 315.43,A -85,B 0,C 180,E1 18519.167,E2 18519.167} C_VEL
LIN {X 0,Y 377.631,Z 315.42,A -85,B 0,C 180,E1 18515.103,E2 18515.103} C_VEL
LIN {X 0,Y 377.635,Z 315.429,A -85,B 0,C 180,E1 18511.191,E2 18511.191} C_VEL
LIN {X 0,Y 377.64,Z 315.434,A -85,B 0,C 180,E1 18507.064,E2 18507.064} C_VEL
LIN {X 0,Y 377.643,Z 315.436,A -85,B 0,C 180,E1 18503.057,E2 18503.057} C_VEL
LIN {X 0,Y 377.645,Z 315.431,A -85,B 0,C 180,E1 18498.958,E2 18498.958} C_VEL
LIN {X 0,Y 377.674,Z 315.59,A -85,B 0,C 180,E1 18494.978,E2 18494.978} C_VEL
LIN {X 0,Y 378.967,Z 318.846,A -85,B 0,C 180,E1 18494.14,E2 18494.14} C_VEL
LIN {X 0,Y 383.475,Z 329.131,A -85,B 0,C 180,E1 18491.78,E2 18491.78} C_VEL
LIN {X 0,Y 388.706,Z 341.635,A -85,B 0,C 180,E1 18489.145,E2 18489.145} C_VEL
LIN {X 0,Y 390.668,Z 346.539,A -85,B 0,C 180,E1 18488.243,E2 18488.243} C_VEL
LIN {X 0,Y 401.854,Z 365.241,A -85,B 0,C 180,E1 18486.428,E2 18486.428} C_VEL
LIN {X 0,Y 408.306,Z 377.391,A -85,B 0,C 180,E1 18485.424,E2 18485.424} C_VEL
LIN {X 0,Y 403.778,Z 562.247,A -85,B 0,C 180,E1 18482.19,E2 18482.19} C_VEL
LIN {X 0,Y 402.985,Z 581.209,A -85,B 0,C 180,E1 18481.604,E2 18481.604} C_VEL
LIN {X 0,Y 401.617,Z 599.757,A -85,B 0,C 180,E1 18480.77,E2 18480.77} C_VEL
LIN {X 0,Y 399.777,Z 617.728,A -85,B 0,C 180,E1 18479.682,E2 18479.682} C_VEL
LIN {X 0,Y 397.538,Z 634.563,A -85,B 0,C 180,E1 18478.382,E2 18478.382} C_VEL
LIN {X 0,Y 395.051,Z 650.399,A -85,B 0,C 180,E1 18476.857,E2 18476.857} C_VEL
LIN {X 0,Y 392.371,Z 665.246,A -85,B 0,C 180,E1 18475.105,E2 18475.105} C_VEL
LIN {X 0,Y 389.631,Z 679.059,A -85,B 0,C 180,E1 18473.117,E2 18473.117} C_VEL
LIN {X 0,Y 386.929,Z 691.753,A -85,B 0,C 180,E1 18470.891,E2 18470.891} C_VEL
LIN {X 0,Y 384.473,Z 702.89,A -85,B 0,C 180,E1 18468.498,E2 18468.498} C_VEL
LIN {X 0,Y 382.352,Z 712.53,A -85,B 0,C 180,E1 18465.936,E2 18465.936} C_VEL
LIN {X 0,Y 381.081,Z 718.294,A -85,B 0,C 180,E1 18464.07,E2 18464.07} C_VEL
LIN {X 0,Y 379.485,Z 721.42,A -85,B 0,C 180,E1 18463.02,E2 18463.02} C_VEL
LIN {X 0,Y 372.358,Z 728.649,A -85,B 0,C 180,E1 18460.368,E2 18460.368} C_VEL
LIN {X 0,Y 370.997,Z 730.832,A -85,B 0,C 180,E1 18459.242,E2 18459.242} C_VEL
LIN {X 0,Y 370.207,Z 734.993,A -85,B 0,C 180,E1 18456.202,E2 18456.202} C_VEL
LIN {X 0,Y 369.783,Z 737.5,A -85,B 0,C 180,E1 18453.1,E2 18453.1} C_VEL
LIN {X 0,Y 369.66,Z 738.341,A -85,B 0,C 180,E1 18450,E2 18450} C_VEL
LIN {X 0,Y 369.78,Z 737.558,A -85,B 0,C 180,E1 18446.9,E2 18446.9} C_VEL
LIN {X 0,Y 370.193,Z 735.114,A -85,B 0,C 180,E1 18443.798,E2 18443.798} C_VEL
LIN {X 0,Y 370.996,Z 730.896,A -85,B 0,C 180,E1 18440.694,E2 18440.694} C_VEL
LIN {X 0,Y 372.169,Z 725.135,A -85,B 0,C 180,E1 18437.747,E2 18437.747} C_VEL
LIN {X 0,Y 373.805,Z 717.823,A -85,B 0,C 180,E1 18434.931,E2 18434.931} C_VEL
LIN {X 0,Y 375.895,Z 708.846,A -85,B 0,C 180,E1 18432.226,E2 18432.226} C_VEL
LIN {X 0,Y 378.28,Z 698.604,A -85,B 0,C 180,E1 18429.742,E2 18429.742} C_VEL
LIN {X 0,Y 380.924,Z 687.124,A -85,B 0,C 180,E1 18427.467,E2 18427.467} C_VEL
LIN {X 0,Y 383.827,Z 673.687,A -85,B 0,C 180,E1 18425.286,E2 18425.286} C_VEL
LIN {X 0,Y 386.627,Z 659.727,A -85,B 0,C 180,E1 18423.424,E2 18423.424} C_VEL
LIN {X 0,Y 389.366,Z 644.318,A -85,B 0,C 180,E1 18421.739,E2 18421.739} C_VEL
LIN {X 0,Y 391.951,Z 627.454,A -85,B 0,C 180,E1 18420.254,E2 18420.254} C_VEL
LIN {X 0,Y 394.089,Z 610.146,A -85,B 0,C 180,E1 18419.044,E2 18419.044} C_VEL
LIN {X 0,Y 395.802,Z 591.756,A -85,B 0,C 180,E1 18418.06,E2 18418.06} C_VEL
LIN {X 0,Y 396.944,Z 572.81,A -85,B 0,C 180,E1 18417.329,E2 18417.329} C_VEL
LIN {X 0,Y 397.505,Z 553.125,A -85,B 0,C 180,E1 18416.846,E2 18416.846} C_VEL
LIN {X 0,Y 401.97,Z 379.768,A -85,B 0,C 180,E1 18413.79,E2 18413.79} C_VEL
LIN {X 0,Y 390.796,Z 359.919,A -85,B 0,C 180,E1 18411.972,E2 18411.972} C_VEL
LIN {X 0,Y 382.406,Z 346.181,A -85,B 0,C 180,E1 18410.473,E2 18410.473} C_VEL
LIN {X 0,Y 376.455,Z 331.742,A -85,B 0,C 180,E1 18407.368,E2 18407.368} C_VEL
LIN {X 0,Y 372.549,Z 323.258,A -85,B 0,C 180,E1 18405.334,E2 18405.334} C_VEL
LIN {X 0,Y 370.815,Z 319.53,A -85,B 0,C 180,E1 18404.396,E2 18404.396} C_VEL
LIN {X 0,Y 369.753,Z 316.556,A -85,B 0,C 180,E1 18403.595,E2 18403.595} C_VEL
LIN {X 0,Y 369.738,Z 316.431,A -85,B 0,C 180,E1 18399.585,E2 18399.585} C_VEL
LIN {X 0,Y 369.731,Z 316.428,A -85,B 0,C 180,E1 18395.515,E2 18395.515} C_VEL
LIN {X 0,Y 369.73,Z 316.43,A -85,B 0,C 180,E1 18391.462,E2 18391.462} C_VEL
LIN {X 0,Y 369.73,Z 316.429,A -85,B 0,C 180,E1 18387.504,E2 18387.504} C_VEL
LIN {X 0,Y 369.722,Z 316.417,A -85,B 0,C 180,E1 18383.425,E2 18383.425} C_VEL
LIN {X 0,Y 369.717,Z 316.405,A -85,B 0,C 180,E1 18379.429,E2 18379.429} C_VEL
LIN {X 0,Y 369.715,Z 316.411,A -85,B 0,C 180,E1 18375.369,E2 18375.369} C_VEL
LIN {X 0,Y 369.716,Z 316.432,A -85,B 0,C 180,E1 18371.387,E2 18371.387} C_VEL
LIN {X 0,Y 369.706,Z 316.414,A -85,B 0,C 180,E1 18367.303,E2 18367.303} C_VEL
LIN {X 0,Y 369.699,Z 316.404,A -85,B 0,C 180,E1 18363.256,E2 18363.256} C_VEL
LIN {X 0,Y 369.701,Z 316.426,A -85,B 0,C 180,E1 18359.226,E2 18359.226} C_VEL
LIN {X 0,Y 369.704,Z 316.426,A -85,B 0,C 180,E1 18355.191,E2 18355.191} C_VEL
LIN {X 0,Y 369.707,Z 316.408,A -85,B 0,C 180,E1 18351.133,E2 18351.133} C_VEL
LIN {X 0,Y 369.707,Z 316.407,A -85,B 0,C 180,E1 18347.029,E2 18347.029} C_VEL
LIN {X 0,Y 369.716,Z 316.424,A -85,B 0,C 180,E1 18343.018,E2 18343.018} C_VEL
LIN {X 0,Y 369.718,Z 316.431,A -85,B 0,C 180,E1 18338.905,E2 18338.905} C_VEL
LIN {X 0,Y 369.722,Z 316.433,A -85,B 0,C 180,E1 18334.876,E2 18334.876} C_VEL
LIN {X 0,Y 369.729,Z 316.433,A -85,B 0,C 180,E1 18330.864,E2 18330.864} C_VEL
LIN {X 0,Y 369.733,Z 316.424,A -85,B 0,C 180,E1 18326.889,E2 18326.889} C_VEL
LIN {X 0,Y 369.758,Z 316.563,A -85,B 0,C 180,E1 18324.927,E2 18324.927} C_VEL
LIN {X 0,Y 370.17,Z 318.223,A -85,B 0,C 180,E1 18324.498,E2 18324.498} C_VEL
LIN {X 0,Y 372.351,Z 322.043,A -85,B 0,C 180,E1 18323.599,E2 18323.599} C_VEL
LIN {X 0,Y 378.902,Z 335.083,A -85,B 0,C 180,E1 18320.877,E2 18320.877} C_VEL
LIN {X 0,Y 386.041,Z 350.283,A -85,B 0,C 180,E1 18318.07,E2 18318.07} C_VEL
LIN {X 0,Y 393.187,Z 367.162,A -85,B 0,C 180,E1 18315.322,E2 18315.322} C_VEL
LIN {X 0,Y 398.556,Z 381.111,A -85,B 0,C 180,E1 18313.295,E2 18313.295} C_VEL
LIN {X 0,Y 402.685,Z 425.422,A -85,B 0,C 180,E1 18311.765,E2 18311.765} C_VEL
LIN {X 0,Y 395.21,Z 634.01,A -85,B 0,C 180,E1 18307.611,E2 18307.611} C_VEL
LIN {X 0,Y 393.553,Z 655.231,A -85,B 0,C 180,E1 18306.969,E2 18306.969} C_VEL
LIN {X 0,Y 391.36,Z 675.145,A -85,B 0,C 180,E1 18306.122,E2 18306.122} C_VEL
LIN {X 0,Y 388.72,Z 695.121,A -85,B 0,C 180,E1 18305,E2 18305} C_VEL
LIN {X 0,Y 385.802,Z 715.033,A -85,B 0,C 180,E1 18303.569,E2 18303.569} C_VEL
LIN {X 0,Y 382.721,Z 734.276,A -85,B 0,C 180,E1 18301.851,E2 18301.851} C_VEL
LIN {X 0,Y 379.775,Z 751.99,A -85,B 0,C 180,E1 18299.927,E2 18299.927} C_VEL
LIN {X 0,Y 376.972,Z 768.772,A -85,B 0,C 180,E1 18297.741,E2 18297.741} C_VEL
LIN {X 0,Y 374.578,Z 783.606,A -85,B 0,C 180,E1 18295.451,E2 18295.451} C_VEL
LIN {X 0,Y 372.495,Z 797.539,A -85,B 0,C 180,E1 18292.905,E2 18292.905} C_VEL
LIN {X 0,Y 370.785,Z 810.714,A -85,B 0,C 180,E1 18290.027,E2 18290.027} C_VEL
LIN {X 0,Y 369.64,Z 821.631,A -85,B 0,C 180,E1 18287.147,E2 18287.147} C_VEL
LIN {X 0,Y 368.991,Z 830.591,A -85,B 0,C 180,E1 18284.275,E2 18284.275} C_VEL
LIN {X 0,Y 368.699,Z 838.139,A -85,B 0,C 180,E1 18281.259,E2 18281.259} C_VEL
LIN {X 0,Y 368.68,Z 843.624,A -85,B 0,C 180,E1 18278.421,E2 18278.421} C_VEL
LIN {X 0,Y 368.803,Z 847.442,A -85,B 0,C 180,E1 18275.601,E2 18275.601} C_VEL
LIN {X 0,Y 368.943,Z 849.809,A -85,B 0,C 180,E1 18272.641,E2 18272.641} C_VEL
LIN {X 0,Y 368.989,Z 850.533,A -85,B 0,C 180,E1 18269.845,E2 18269.845} C_VEL
LIN {X 0,Y 368.929,Z 849.649,A -85,B 0,C 180,E1 18267.048,E2 18267.048} C_VEL
LIN {X 0,Y 368.783,Z 847.073,A -85,B 0,C 180,E1 18264.087,E2 18264.087} C_VEL
LIN {X 0,Y 368.677,Z 843.092,A -85,B 0,C 180,E1 18261.265,E2 18261.265} C_VEL
LIN {X 0,Y 368.719,Z 837.108,A -85,B 0,C 180,E1 18258.266,E2 18258.266} C_VEL
LIN {X 0,Y 369.076,Z 829.228,A -85,B 0,C 180,E1 18255.247,E2 18255.247} C_VEL
LIN {X 0,Y 369.794,Z 819.913,A -85,B 0,C 180,E1 18252.373,E2 18252.373} C_VEL
LIN {X 0,Y 371.027,Z 808.611,A -85,B 0,C 180,E1 18249.493,E2 18249.493} C_VEL
LIN {X 0,Y 372.723,Z 795.847,A -85,B 0,C 180,E1 18246.776,E2 18246.776} C_VEL
LIN {X 0,Y 374.873,Z 781.648,A -85,B 0,C 180,E1 18244.231,E2 18244.231} C_VEL
LIN {X 0,Y 377.437,Z 765.979,A -85,B 0,C 180,E1 18241.867,E2 18241.867} C_VEL
LIN {X 0,Y 380.316,Z 748.703,A -85,B 0,C 180,E1 18239.685,E2 18239.685} C_VEL
LIN {X 0,Y 383.337,Z 730.572,A -85,B 0,C 180,E1 18237.79,E2 18237.79} C_VEL
LIN {X 0,Y 386.269,Z 711.874,A -85,B 0,C 180,E1 18236.185,E2 18236.185} C_VEL
LIN {X 0,Y 389.045,Z 692.678,A -85,B 0,C 180,E1 18234.853,E2 18234.853} C_VEL
LIN {X 0,Y 391.54,Z 673.367,A -85,B 0,C 180,E1 18233.799,E2 18233.799} C_VEL
LIN {X 0,Y 393.829,Z 651.904,A -85,B 0,C 180,E1 18232.924,E2 18232.924} C_VEL
LIN {X 0,Y 395.373,Z 629.735,A -85,B 0,C 180,E1 18232.299,E2 18232.299} C_VEL
LIN {X 0,Y 402.659,Z 424.289,A -85,B 0,C 180,E1 18228.22,E2 18228.22} C_VEL
LIN {X 0,Y 398.425,Z 380.897,A -85,B 0,C 180,E1 18226.699,E2 18226.699} C_VEL
LIN {X 0,Y 391.232,Z 362.281,A -85,B 0,C 180,E1 18223.936,E2 18223.936} C_VEL
LIN {X 0,Y 383.727,Z 345.139,A -85,B 0,C 180,E1 18221.043,E2 18221.043} C_VEL
LIN {X 0,Y 377.601,Z 332.574,A -85,B 0,C 180,E1 18218.637,E2 18218.637} C_VEL
LIN {X 0,Y 373.7,Z 324.765,A -85,B 0,C 180,E1 18217.013,E2 18217.013} C_VEL
LIN {X 0,Y 371.587,Z 320.616,A -85,B 0,C 180,E1 18216.106,E2 18216.106} C_VEL
LIN {X 0,Y 369.853,Z 317.138,A -85,B 0,C 180,E1 18215.32,E2 18215.32} C_VEL
LIN {X 0,Y 369.741,Z 316.427,A -85,B 0,C 180,E1 18214.98,E2 18214.98} C_VEL
LIN {X 0,Y 369.745,Z 316.412,A -85,B 0,C 180,E1 18210.917,E2 18210.917} C_VEL
LIN {X 0,Y 369.741,Z 316.412,A -85,B 0,C 180,E1 18206.828,E2 18206.828} C_VEL
LIN {X 0,Y 369.745,Z 316.408,A -85,B 0,C 180,E1 18202.749,E2 18202.749} C_VEL
LIN {X 0,Y 369.732,Z 316.407,A -85,B 0,C 180,E1 18198.608,E2 18198.608} C_VEL
LIN {X 0,Y 369.73,Z 316.41,A -85,B 0,C 180,E1 18194.509,E2 18194.509} C_VEL
LIN {X 0,Y 369.719,Z 316.429,A -85,B 0,C 180,E1 18190.439,E2 18190.439} C_VEL
LIN {X 0,Y 369.718,Z 316.424,A -85,B 0,C 180,E1 18186.366,E2 18186.366} C_VEL
LIN {X 0,Y 369.707,Z 316.406,A -85,B 0,C 180,E1 18182.325,E2 18182.325} C_VEL
LIN {X 0,Y 369.704,Z 316.414,A -85,B 0,C 180,E1 18178.295,E2 18178.295} C_VEL
LIN {X 0,Y 369.7,Z 316.434,A -85,B 0,C 180,E1 18174.101,E2 18174.101} C_VEL
LIN {X 0,Y 369.709,Z 316.411,A -85,B 0,C 180,E1 18170.19,E2 18170.19} C_VEL
LIN {X 0,Y 369.708,Z 316.404,A -85,B 0,C 180,E1 18166.072,E2 18166.072} C_VEL
LIN {X 0,Y 369.717,Z 316.423,A -85,B 0,C 180,E1 18162.043,E2 18162.043} C_VEL
LIN {X 0,Y 369.717,Z 316.433,A -85,B 0,C 180,E1 18157.919,E2 18157.919} C_VEL
LIN {X 0,Y 369.718,Z 316.419,A -85,B 0,C 180,E1 18153.844,E2 18153.844} C_VEL
LIN {X 0,Y 369.731,Z 316.411,A -85,B 0,C 180,E1 18149.922,E2 18149.922} C_VEL
LIN {X 0,Y 369.73,Z 316.412,A -85,B 0,C 180,E1 18145.842,E2 18145.842} C_VEL
LIN {X 0,Y 369.73,Z 316.415,A -85,B 0,C 180,E1 18141.736,E2 18141.736} C_VEL
LIN {X 0,Y 369.732,Z 316.419,A -85,B 0,C 180,E1 18137.672,E2 18137.672} C_VEL
LIN {X 0,Y 369.783,Z 316.727,A -85,B 0,C 180,E1 18136.195,E2 18136.195} C_VEL
LIN {X 0,Y 371.162,Z 320.086,A -85,B 0,C 180,E1 18135.323,E2 18135.323} C_VEL
LIN {X 0,Y 375.606,Z 329.93,A -85,B 0,C 180,E1 18132.941,E2 18132.941} C_VEL
LIN {X 0,Y 381.065,Z 342.824,A -85,B 0,C 180,E1 18130.105,E2 18130.105} C_VEL
LIN {X 0,Y 382.832,Z 347.151,A -85,B 0,C 180,E1 18129.28,E2 18129.28} C_VEL
LIN {X 0,Y 394.094,Z 365.545,A -85,B 0,C 180,E1 18127.368,E2 18127.368} C_VEL
LIN {X 0,Y 402.008,Z 380.162,A -85,B 0,C 180,E1 18126.09,E2 18126.09} C_VEL
LIN {X 0,Y 397.256,Z 562.922,A -85,B 0,C 180,E1 18122.846,E2 18122.846} C_VEL
LIN {X 0,Y 396.432,Z 581.766,A -85,B 0,C 180,E1 18122.258,E2 18122.258} C_VEL
LIN {X 0,Y 395.024,Z 600.147,A -85,B 0,C 180,E1 18121.426,E2 18121.426} C_VEL
LIN {X 0,Y 393.223,Z 617.149,A -85,B 0,C 180,E1 18120.397,E2 18120.397} C_VEL
LIN {X 0,Y 391.012,Z 633.44,A -85,B 0,C 180,E1 18119.151,E2 18119.151} C_VEL
LIN {X 0,Y 388.517,Z 648.98,A -85,B 0,C 180,E1 18117.678,E2 18117.678} C_VEL
LIN {X 0,Y 385.67,Z 664.336,A -85,B 0,C 180,E1 18115.893,E2 18115.893} C_VEL
LIN {X 0,Y 382.777,Z 678.445,A -85,B 0,C 180,E1 18113.883,E2 18113.883} C_VEL
LIN {X 0,Y 380.077,Z 690.644,A -85,B 0,C 180,E1 18111.772,E2 18111.772} C_VEL
LIN {X 0,Y 377.41,Z 702.183,A -85,B 0,C 180,E1 18109.338,E2 18109.338} C_VEL
LIN {X 0,Y 375.092,Z 712.176,A -85,B 0,C 180,E1 18106.731,E2 18106.731} C_VEL
LIN {X 0,Y 373.137,Z 720.642,A -85,B 0,C 180,E1 18103.955,E2 18103.955} C_VEL
LIN {X 0,Y 371.641,Z 727.555,A -85,B 0,C 180,E1 18101.012,E2 18101.012} C_VEL
LIN {X 0,Y 370.997,Z 730.832,A -85,B 0,C 180,E1 18099.242,E2 18099.242} C_VEL
LIN {X 0,Y 369.69,Z 732.861,A -85,B 0,C 180,E1 18098.1,E2 18098.1} C_VEL
LIN {X 0,Y 364.253,Z 736.462,A -85,B 0,C 180,E1 18095.777,E2 18095.777} C_VEL
LIN {X 0,Y 362.158,Z 737.879,A -85,B 0,C 180,E1 18094.424,E2 18094.424} C_VEL
LIN {X 0,Y 361.958,Z 738.178,A -85,B 0,C 180,E1 18093.987,E2 18093.987} C_VEL
LIN {X 0,Y 361.753,Z 739.441,A -85,B 0,C 180,E1 18090.792,E2 18090.792} C_VEL
LIN {X 0,Y 361.816,Z 739.062,A -85,B 0,C 180,E1 18087.624,E2 18087.624} C_VEL
LIN {X 0,Y 362.17,Z 737.043,A -85,B 0,C 180,E1 18084.455,E2 18084.455} C_VEL
LIN {X 0,Y 362.911,Z 733.295,A -85,B 0,C 180,E1 18081.285,E2 18081.285} C_VEL
LIN {X 0,Y 364.039,Z 728.011,A -85,B 0,C 180,E1 18078.274,E2 18078.274} C_VEL
LIN {X 0,Y 365.698,Z 720.873,A -85,B 0,C 180,E1 18075.27,E2 18075.27} C_VEL
LIN {X 0,Y 367.704,Z 712.688,A -85,B 0,C 180,E1 18072.596,E2 18072.596} C_VEL
LIN {X 0,Y 370.188,Z 702.54,A -85,B 0,C 180,E1 18069.94,E2 18069.94} C_VEL
LIN {X 0,Y 373.036,Z 690.826,A -85,B 0,C 180,E1 18067.463,E2 18067.463} C_VEL
LIN {X 0,Y 375.895,Z 678.427,A -85,B 0,C 180,E1 18065.317,E2 18065.317} C_VEL
LIN {X 0,Y 378.848,Z 664.599,A -85,B 0,C 180,E1 18063.343,E2 18063.343} C_VEL
LIN {X 0,Y 381.823,Z 649.137,A -85,B 0,C 180,E1 18061.538,E2 18061.538} C_VEL
LIN {X 0,Y 384.454,Z 633.384,A -85,B 0,C 180,E1 18060.045,E2 18060.045} C_VEL
LIN {X 0,Y 386.892,Z 615.704,A -85,B 0,C 180,E1 18058.706,E2 18058.706} C_VEL
LIN {X 0,Y 388.777,Z 597.903,A -85,B 0,C 180,E1 18057.662,E2 18057.662} C_VEL
LIN {X 0,Y 390.173,Z 578.929,A -85,B 0,C 180,E1 18056.843,E2 18056.843} C_VEL
LIN {X 0,Y 390.918,Z 559.61,A -85,B 0,C 180,E1 18056.286,E2 18056.286} C_VEL
LIN {X 0,Y 395.719,Z 382.656,A -85,B 0,C 180,E1 18053.102,E2 18053.102} C_VEL
LIN {X 0,Y 385.088,Z 363.871,A -85,B 0,C 180,E1 18051.312,E2 18051.312} C_VEL
LIN {X 0,Y 374.883,Z 347.475,A -85,B 0,C 180,E1 18049.476,E2 18049.476} C_VEL
LIN {X 0,Y 368.778,Z 333.08,A -85,B 0,C 180,E1 18046.263,E2 18046.263} C_VEL
LIN {X 0,Y 364.779,Z 324.491,A -85,B 0,C 180,E1 18044.101,E2 18044.101} C_VEL
LIN {X 0,Y 363.332,Z 321.242,A -85,B 0,C 180,E1 18043.254,E2 18043.254} C_VEL
LIN {X 0,Y 361.83,Z 317.634,A -85,B 0,C 180,E1 18042.249,E2 18042.249} C_VEL
LIN {X 0,Y 361.794,Z 317.402,A -85,B 0,C 180,E1 18038.247,E2 18038.247} C_VEL
LIN {X 0,Y 361.794,Z 317.399,A -85,B 0,C 180,E1 18034.126,E2 18034.126} C_VEL
LIN {X 0,Y 361.798,Z 317.397,A -85,B 0,C 180,E1 18030.014,E2 18030.014} C_VEL
LIN {X 0,Y 361.795,Z 317.401,A -85,B 0,C 180,E1 18025.891,E2 18025.891} C_VEL
LIN {X 0,Y 361.807,Z 317.415,A -85,B 0,C 180,E1 18021.735,E2 18021.735} C_VEL
LIN {X 0,Y 361.789,Z 317.414,A -85,B 0,C 180,E1 18017.532,E2 18017.532} C_VEL
LIN {X 0,Y 361.777,Z 317.395,A -85,B 0,C 180,E1 18013.392,E2 18013.392} C_VEL
LIN {X 0,Y 361.771,Z 317.393,A -85,B 0,C 180,E1 18009.375,E2 18009.375} C_VEL
LIN {X 0,Y 361.774,Z 317.42,A -85,B 0,C 180,E1 18005.392,E2 18005.392} C_VEL
LIN {X 0,Y 361.762,Z 317.407,A -85,B 0,C 180,E1 18001.267,E2 18001.267} C_VEL
LIN {X 0,Y 361.757,Z 317.392,A -85,B 0,C 180,E1 17997.149,E2 17997.149} C_VEL
LIN {X 0,Y 361.758,Z 317.404,A -85,B 0,C 180,E1 17993.015,E2 17993.015} C_VEL
LIN {X 0,Y 361.766,Z 317.422,A -85,B 0,C 180,E1 17989.006,E2 17989.006} C_VEL
LIN {X 0,Y 361.767,Z 317.41,A -85,B 0,C 180,E1 17984.942,E2 17984.942} C_VEL
LIN {X 0,Y 361.773,Z 317.4,A -85,B 0,C 180,E1 17980.941,E2 17980.941} C_VEL
LIN {X 0,Y 361.779,Z 317.398,A -85,B 0,C 180,E1 17976.893,E2 17976.893} C_VEL
LIN {X 0,Y 361.784,Z 317.4,A -85,B 0,C 180,E1 17972.858,E2 17972.858} C_VEL
LIN {X 0,Y 361.793,Z 317.401,A -85,B 0,C 180,E1 17968.883,E2 17968.883} C_VEL
LIN {X 0,Y 361.809,Z 317.689,A -85,B 0,C 180,E1 17966.283,E2 17966.283} C_VEL
LIN {X 0,Y 363.225,Z 321.045,A -85,B 0,C 180,E1 17965.455,E2 17965.455} C_VEL
LIN {X 0,Y 364.353,Z 322.737,A -85,B 0,C 180,E1 17965.003,E2 17965.003} C_VEL
LIN {X 0,Y 366.44,Z 326.654,A -85,B 0,C 180,E1 17964.081,E2 17964.081} C_VEL
LIN {X 0,Y 373.538,Z 341.123,A -85,B 0,C 180,E1 17961.022,E2 17961.022} C_VEL
LIN {X 0,Y 380.254,Z 355.639,A -85,B 0,C 180,E1 17958.299,E2 17958.299} C_VEL
LIN {X 0,Y 387.27,Z 372.531,A -85,B 0,C 180,E1 17955.496,E2 17955.496} C_VEL
LIN {X 0,Y 390.404,Z 380.571,A -85,B 0,C 180,E1 17954.316,E2 17954.316} C_VEL
LIN {X 0,Y 392.72,Z 385.25,A -85,B 0,C 180,E1 17953.91,E2 17953.91} C_VEL
LIN {X 0,Y 396.383,Z 426.827,A -85,B 0,C 180,E1 17952.457,E2 17952.457} C_VEL
LIN {X 0,Y 388.623,Z 633.809,A -85,B 0,C 180,E1 17948.28,E2 17948.28} C_VEL
LIN {X 0,Y 386.828,Z 655.575,A -85,B 0,C 180,E1 17947.604,E2 17947.604} C_VEL
LIN {X 0,Y 384.509,Z 675.463,A -85,B 0,C 180,E1 17946.731,E2 17946.731} C_VEL
LIN {X 0,Y 381.867,Z 694.456,A -85,B 0,C 180,E1 17945.639,E2 17945.639} C_VEL
LIN {X 0,Y 378.833,Z 714.109,A -85,B 0,C 180,E1 17944.205,E2 17944.205} C_VEL
LIN {X 0,Y 375.571,Z 733.516,A -85,B 0,C 180,E1 17942.443,E2 17942.443} C_VEL
LIN {X 0,Y 372.347,Z 751.824,A -85,B 0,C 180,E1 17940.408,E2 17940.408} C_VEL
LIN {X 0,Y 369.411,Z 768.447,A -85,B 0,C 180,E1 17938.183,E2 17938.183} C_VEL
LIN {X 0,Y 366.894,Z 783.145,A -85,B 0,C 180,E1 17935.85,E2 17935.85} C_VEL
LIN {X 0,Y 364.705,Z 796.986,A -85,B 0,C 180,E1 17933.252,E2 17933.252} C_VEL
LIN {X 0,Y 362.907,Z 810.07,A -85,B 0,C 180,E1 17930.312,E2 17930.312} C_VEL
LIN {X 0,Y 361.65,Z 821.465,A -85,B 0,C 180,E1 17927.206,E2 17927.206} C_VEL
LIN {X 0,Y 360.973,Z 830.671,A -85,B 0,C 180,E1 17924.108,E2 17924.108} C_VEL
LIN {X 0,Y 360.722,Z 837.916,A -85,B 0,C 180,E1 17921.026,E2 17921.026} C_VEL
LIN {X 0,Y 360.753,Z 843.342,A -85,B 0,C 180,E1 17917.965,E2 17917.965} C_VEL
LIN {X 0,Y 360.901,Z 846.9,A -85,B 0,C 180,E1 17915.086,E2 17915.086} C_VEL
LIN {X 0,Y 361.035,Z 848.838,A -85,B 0,C 180,E1 17912.222,E2 17912.222} C_VEL
LIN {X 0,Y 361.073,Z 849.256,A -85,B 0,C 180,E1 17909.365,E2 17909.365} C_VEL
LIN {X 0,Y 360.979,Z 848.194,A -85,B 0,C 180,E1 17906.506,E2 17906.506} C_VEL
LIN {X 0,Y 360.83,Z 845.488,A -85,B 0,C 180,E1 17903.636,E2 17903.636} C_VEL
LIN {X 0,Y 360.721,Z 840.992,A -85,B 0,C 180,E1 17900.588,E2 17900.588} C_VEL
LIN {X 0,Y 360.775,Z 835.116,A -85,B 0,C 180,E1 17897.679,E2 17897.679} C_VEL
LIN {X 0,Y 361.203,Z 827.04,A -85,B 0,C 180,E1 17894.589,E2 17894.589} C_VEL
LIN {X 0,Y 362.032,Z 817.468,A -85,B 0,C 180,E1 17891.649,E2 17891.649} C_VEL
LIN {X 0,Y 363.331,Z 806.583,A -85,B 0,C 180,E1 17888.87,E2 17888.87} C_VEL
LIN {X 0,Y 365.194,Z 793.65,A -85,B 0,C 180,E1 17886.097,E2 17886.097} C_VEL
LIN {X 0,Y 367.529,Z 779.26,A -85,B 0,C 180,E1 17883.503,E2 17883.503} C_VEL
LIN {X 0,Y 370.249,Z 763.693,A -85,B 0,C 180,E1 17881.143,E2 17881.143} C_VEL
LIN {X 0,Y 373.268,Z 746.52,A -85,B 0,C 180,E1 17878.961,E2 17878.961} C_VEL
LIN {X 0,Y 376.417,Z 728.601,A -85,B 0,C 180,E1 17877.074,E2 17877.074} C_VEL
LIN {X 0,Y 379.598,Z 709.338,A -85,B 0,C 180,E1 17875.416,E2 17875.416} C_VEL
LIN {X 0,Y 382.536,Z 689.796,A -85,B 0,C 180,E1 17874.072,E2 17874.072} C_VEL
LIN {X 0,Y 385.131,Z 670.054,A -85,B 0,C 180,E1 17873.012,E2 17873.012} C_VEL
LIN {X 0,Y 387.372,Z 649.543,A -85,B 0,C 180,E1 17872.197,E2 17872.197} C_VEL
LIN {X 0,Y 388.855,Z 628.164,A -85,B 0,C 180,E1 17871.598,E2 17871.598} C_VEL
LIN {X 0,Y 396.355,Z 425.215,A -85,B 0,C 180,E1 17867.517,E2 17867.517} C_VEL
LIN {X 0,Y 392.46,Z 384.426,A -85,B 0,C 180,E1 17866.057,E2 17866.057} C_VEL
LIN {X 0,Y 389.67,Z 378.987,A -85,B 0,C 180,E1 17865.506,E2 17865.506} C_VEL
LIN {X 0,Y 383.271,Z 362.639,A -85,B 0,C 180,E1 17862.912,E2 17862.912} C_VEL
LIN {X 0,Y 376.067,Z 346.399,A -85,B 0,C 180,E1 17860.032,E2 17860.032} C_VEL
LIN {X 0,Y 370.219,Z 334.377,A -85,B 0,C 180,E1 17857.615,E2 17857.615} C_VEL
LIN {X 0,Y 365.908,Z 325.96,A -85,B 0,C 180,E1 17855.753,E2 17855.753} C_VEL
LIN {X 0,Y 363.974,Z 321.946,A -85,B 0,C 180,E1 17854.847,E2 17854.847} C_VEL
LIN {X 0,Y 362.14,Z 318.988,A -85,B 0,C 180,E1 17854.079,E2 17854.079} C_VEL
LIN {X 0,Y 361.774,Z 317.425,A -85,B 0,C 180,E1 17853.623,E2 17853.623} C_VEL
LIN {X 0,Y 361.774,Z 317.422,A -85,B 0,C 180,E1 17849.468,E2 17849.468} C_VEL
LIN {X 0,Y 361.772,Z 317.424,A -85,B 0,C 180,E1 17845.347,E2 17845.347} C_VEL
LIN {X 0,Y 361.767,Z 317.419,A -85,B 0,C 180,E1 17841.349,E2 17841.349} C_VEL
LIN {X 0,Y 361.756,Z 317.407,A -85,B 0,C 180,E1 17837.367,E2 17837.367} C_VEL
LIN {X 0,Y 361.75,Z 317.396,A -85,B 0,C 180,E1 17833.374,E2 17833.374} C_VEL
LIN {X 0,Y 361.747,Z 317.404,A -85,B 0,C 180,E1 17829.352,E2 17829.352} C_VEL
LIN {X 0,Y 361.743,Z 317.425,A -85,B 0,C 180,E1 17825.392,E2 17825.392} C_VEL
LIN {X 0,Y 361.738,Z 317.411,A -85,B 0,C 180,E1 17821.267,E2 17821.267} C_VEL
LIN {X 0,Y 361.734,Z 317.395,A -85,B 0,C 180,E1 17817.148,E2 17817.148} C_VEL
LIN {X 0,Y 361.738,Z 317.416,A -85,B 0,C 180,E1 17813.174,E2 17813.174} C_VEL
LIN {X 0,Y 361.749,Z 317.422,A -85,B 0,C 180,E1 17809.005,E2 17809.005} C_VEL
LIN {X 0,Y 361.751,Z 317.398,A -85,B 0,C 180,E1 17804.941,E2 17804.941} C_VEL
LIN {X 0,Y 361.755,Z 317.398,A -85,B 0,C 180,E1 17800.949,E2 17800.949} C_VEL
LIN {X 0,Y 361.76,Z 317.414,A -85,B 0,C 180,E1 17796.891,E2 17796.891} C_VEL
LIN {X 0,Y 361.765,Z 317.423,A -85,B 0,C 180,E1 17792.864,E2 17792.864} C_VEL
LIN {X 0,Y 361.764,Z 317.417,A -85,B 0,C 180,E1 17788.879,E2 17788.879} C_VEL
LIN {X 0,Y 361.772,Z 317.415,A -85,B 0,C 180,E1 17784.716,E2 17784.716} C_VEL
LIN {X 0,Y 361.776,Z 317.417,A -85,B 0,C 180,E1 17780.699,E2 17780.699} C_VEL
LIN {X 0,Y 361.828,Z 317.682,A -85,B 0,C 180,E1 17777.603,E2 17777.603} C_VEL
LIN {X 0,Y 363.111,Z 320.945,A -85,B 0,C 180,E1 17776.713,E2 17776.713} C_VEL
LIN {X 0,Y 364.066,Z 322.79,A -85,B 0,C 180,E1 17776.204,E2 17776.204} C_VEL
LIN {X 0,Y 369.244,Z 334.106,A -85,B 0,C 180,E1 17773.359,E2 17773.359} C_VEL
LIN {X 0,Y 374.977,Z 347.675,A -85,B 0,C 180,E1 17770.386,E2 17770.386} C_VEL
LIN {X 0,Y 387.256,Z 367.582,A -85,B 0,C 180,E1 17768.198,E2 17768.198} C_VEL
LIN {X 0,Y 395.768,Z 382.959,A -85,B 0,C 180,E1 17766.776,E2 17766.776} C_VEL
LIN {X 0,Y 390.787,Z 563.632,A -85,B 0,C 180,E1 17763.522,E2 17763.522} C_VEL
LIN {X 0,Y 389.925,Z 582.444,A -85,B 0,C 180,E1 17762.929,E2 17762.929} C_VEL
LIN {X 0,Y 388.497,Z 600.381,A -85,B 0,C 180,E1 17762.112,E2 17762.112} C_VEL
LIN {X 0,Y 386.602,Z 617.669,A -85,B 0,C 180,E1 17761.061,E2 17761.061} C_VEL
LIN {X 0,Y 384.298,Z 634.059,A -85,B 0,C 180,E1 17759.797,E2 17759.797} C_VEL
LIN {X 0,Y 381.56,Z 650.388,A -85,B 0,C 180,E1 17758.228,E2 17758.228} C_VEL
LIN {X 0,Y 378.602,Z 665.622,A -85,B 0,C 180,E1 17756.422,E2 17756.422} C_VEL
LIN {X 0,Y 375.567,Z 679.75,A -85,B 0,C 180,E1 17754.371,E2 17754.371} C_VEL
LIN {X 0,Y 372.742,Z 691.919,A -85,B 0,C 180,E1 17752.223,E2 17752.223} C_VEL
LIN {X 0,Y 369.945,Z 703.438,A -85,B 0,C 180,E1 17749.745,E2 17749.745} C_VEL
LIN {X 0,Y 367.507,Z 713.414,A -85,B 0,C 180,E1 17747.087,E2 17747.087} C_VEL
LIN {X 0,Y 365.445,Z 721.869,A -85,B 0,C 180,E1 17744.255,E2 17744.255} C_VEL
LIN {X 0,Y 363.93,Z 728.45,A -85,B 0,C 180,E1 17741.409,E2 17741.409} C_VEL
LIN {X 0,Y 362.838,Z 733.614,A -85,B 0,C 180,E1 17738.393,E2 17738.393} C_VEL
LIN {X 0,Y 362.132,Z 737.234,A -85,B 0,C 180,E1 17735.228,E2 17735.228} C_VEL
LIN {X 0,Y 361.958,Z 738.178,A -85,B 0,C 180,E1 17733.987,E2 17733.987} C_VEL
LIN {X 0,Y 360.846,Z 739.026,A -85,B 0,C 180,E1 17732.776,E2 17732.776} C_VEL
LIN {X 0,Y 354.676,Z 740.6,A -85,B 0,C 180,E1 17729.615,E2 17729.615} C_VEL
LIN {X 0,Y 353.866,Z 740.566,A -85,B 0,C 180,E1 17728.451,E2 17728.451} C_VEL
LIN {X 0,Y 354.168,Z 738.956,A -85,B 0,C 180,E1 17725.142,E2 17725.142} C_VEL
LIN {X 0,Y 354.843,Z 735.653,A -85,B 0,C 180,E1 17721.901,E2 17721.901} C_VEL
LIN {X 0,Y 355.983,Z 730.512,A -85,B 0,C 180,E1 17718.662,E2 17718.662} C_VEL
LIN {X 0,Y 357.614,Z 723.781,A -85,B 0,C 180,E1 17715.592,E2 17715.592} C_VEL
LIN {X 0,Y 359.742,Z 715.516,A -85,B 0,C 180,E1 17712.699,E2 17712.699} C_VEL
LIN {X 0,Y 362.259,Z 705.753,A -85,B 0,C 180,E1 17709.987,E2 17709.987} C_VEL
LIN {X 0,Y 365.146,Z 694.482,A -85,B 0,C 180,E1 17707.459,E2 17707.459} C_VEL
LIN {X 0,Y 368.067,Z 682.609,A -85,B 0,C 180,E1 17705.271,E2 17705.271} C_VEL
LIN {X 0,Y 371.207,Z 668.841,A -85,B 0,C 180,E1 17703.182,E2 17703.182} C_VEL
LIN {X 0,Y 374.271,Z 654.067,A -85,B 0,C 180,E1 17701.346,E2 17701.346} C_VEL
LIN {X 0,Y 377.109,Z 638.352,A -85,B 0,C 180,E1 17699.752,E2 17699.752} C_VEL
LIN {X 0,Y 379.653,Z 621.703,A -85,B 0,C 180,E1 17698.394,E2 17698.394} C_VEL
LIN {X 0,Y 381.841,Z 603.378,A -85,B 0,C 180,E1 17697.224,E2 17697.224} C_VEL
LIN {X 0,Y 383.453,Z 584.426,A -85,B 0,C 180,E1 17696.325,E2 17696.325} C_VEL
LIN {X 0,Y 384.412,Z 565.234,A -85,B 0,C 180,E1 17695.699,E2 17695.699} C_VEL
LIN {X 0,Y 386.262,Z 495.829,A -85,B 0,C 180,E1 17694.403,E2 17694.403} C_VEL
LIN {X 0,Y 389.523,Z 385.592,A -85,B 0,C 180,E1 17692.393,E2 17692.393} C_VEL
LIN {X 0,Y 378.787,Z 366.622,A -85,B 0,C 180,E1 17690.513,E2 17690.513} C_VEL
LIN {X 0,Y 367.094,Z 348.215,A -85,B 0,C 180,E1 17688.32,E2 17688.32} C_VEL
LIN {X 0,Y 361.38,Z 334.825,A -85,B 0,C 180,E1 17685.209,E2 17685.209} C_VEL
LIN {X 0,Y 357.156,Z 326.047,A -85,B 0,C 180,E1 17682.866,E2 17682.866} C_VEL
LIN {X 0,Y 355.397,Z 322.186,A -85,B 0,C 180,E1 17681.797,E2 17681.797} C_VEL
LIN {X 0,Y 353.872,Z 318.649,A -85,B 0,C 180,E1 17680.745,E2 17680.745} C_VEL
LIN {X 0,Y 353.833,Z 318.398,A -85,B 0,C 180,E1 17676.804,E2 17676.804} C_VEL
LIN {X 0,Y 353.83,Z 318.399,A -85,B 0,C 180,E1 17672.641,E2 17672.641} C_VEL
LIN {X 0,Y 353.83,Z 318.393,A -85,B 0,C 180,E1 17668.502,E2 17668.502} C_VEL
LIN {X 0,Y 353.828,Z 318.384,A -85,B 0,C 180,E1 17664.367,E2 17664.367} C_VEL
LIN {X 0,Y 353.826,Z 318.385,A -85,B 0,C 180,E1 17660.256,E2 17660.256} C_VEL
LIN {X 0,Y 353.831,Z 318.4,A -85,B 0,C 180,E1 17656.077,E2 17656.077} C_VEL
LIN {X 0,Y 353.833,Z 318.407,A -85,B 0,C 180,E1 17651.905,E2 17651.905} C_VEL
LIN {X 0,Y 353.848,Z 318.382,A -85,B 0,C 180,E1 17647.632,E2 17647.632} C_VEL
LIN {X 0,Y 353.827,Z 318.38,A -85,B 0,C 180,E1 17643.402,E2 17643.402} C_VEL
LIN {X 0,Y 353.82,Z 318.403,A -85,B 0,C 180,E1 17639.191,E2 17639.191} C_VEL
LIN {X 0,Y 353.813,Z 318.409,A -85,B 0,C 180,E1 17634.975,E2 17634.975} C_VEL
LIN {X 0,Y 353.815,Z 318.387,A -85,B 0,C 180,E1 17630.895,E2 17630.895} C_VEL
LIN {X 0,Y 353.815,Z 318.384,A -85,B 0,C 180,E1 17626.768,E2 17626.768} C_VEL
LIN {X 0,Y 353.821,Z 318.397,A -85,B 0,C 180,E1 17622.74,E2 17622.74} C_VEL
LIN {X 0,Y 353.824,Z 318.407,A -85,B 0,C 180,E1 17618.621,E2 17618.621} C_VEL
LIN {X 0,Y 353.829,Z 318.411,A -85,B 0,C 180,E1 17614.563,E2 17614.563} C_VEL
LIN {X 0,Y 353.827,Z 318.405,A -85,B 0,C 180,E1 17610.362,E2 17610.362} C_VEL
LIN {X 0,Y 353.867,Z 318.641,A -85,B 0,C 180,E1 17607.844,E2 17607.844} C_VEL
LIN {X 0,Y 355.335,Z 322.13,A -85,B 0,C 180,E1 17606.915,E2 17606.915} C_VEL
LIN {X 0,Y 356.543,Z 324.006,A -85,B 0,C 180,E1 17606.393,E2 17606.393} C_VEL
LIN {X 0,Y 359.087,Z 328.882,A -85,B 0,C 180,E1 17605.194,E2 17605.194} C_VEL
LIN {X 0,Y 363.891,Z 338.413,A -85,B 0,C 180,E1 17603.006,E2 17603.006} C_VEL
LIN {X 0,Y 370.158,Z 351.303,A -85,B 0,C 180,E1 17600.337,E2 17600.337} C_VEL
LIN {X 0,Y 377.444,Z 368.019,A -85,B 0,C 180,E1 17597.301,E2 17597.301} C_VEL
LIN {X 0,Y 382.211,Z 379.875,A -85,B 0,C 180,E1 17595.407,E2 17595.407} C_VEL
LIN {X 0,Y 386.858,Z 388.891,A -85,B 0,C 180,E1 17594.566,E2 17594.566} C_VEL
LIN {X 0,Y 390.151,Z 428.02,A -85,B 0,C 180,E1 17593.175,E2 17593.175} C_VEL
LIN {X 0,Y 382.1,Z 633.428,A -85,B 0,C 180,E1 17588.976,E2 17588.976} C_VEL
LIN {X 0,Y 380.185,Z 655.538,A -85,B 0,C 180,E1 17588.273,E2 17588.273} C_VEL
LIN {X 0,Y 377.611,Z 676.539,A -85,B 0,C 180,E1 17587.325,E2 17587.325} C_VEL
LIN {X 0,Y 374.68,Z 696.317,A -85,B 0,C 180,E1 17586.138,E2 17586.138} C_VEL
LIN {X 0,Y 371.564,Z 715.319,A -85,B 0,C 180,E1 17584.689,E2 17584.689} C_VEL
LIN {X 0,Y 368.342,Z 733.432,A -85,B 0,C 180,E1 17582.99,E2 17582.99} C_VEL
LIN {X 0,Y 365.059,Z 751.037,A -85,B 0,C 180,E1 17580.989,E2 17580.989} C_VEL
LIN {X 0,Y 361.872,Z 768.129,A -85,B 0,C 180,E1 17578.644,E2 17578.644} C_VEL
LIN {X 0,Y 359.067,Z 783.6,A -85,B 0,C 180,E1 17576.101,E2 17576.101} C_VEL
LIN {X 0,Y 356.801,Z 797.175,A -85,B 0,C 180,E1 17573.448,E2 17573.448} C_VEL
LIN {X 0,Y 355.032,Z 809.393,A -85,B 0,C 180,E1 17570.611,E2 17570.611} C_VEL
LIN {X 0,Y 353.768,Z 820.169,A -85,B 0,C 180,E1 17567.602,E2 17567.602} C_VEL
LIN {X 0,Y 353.035,Z 829.399,A -85,B 0,C 180,E1 17564.432,E2 17564.432} C_VEL
LIN {X 0,Y 352.76,Z 836.669,A -85,B 0,C 180,E1 17561.277,E2 17561.277} C_VEL
LIN {X 0,Y 352.798,Z 842.114,A -85,B 0,C 180,E1 17558.146,E2 17558.146} C_VEL
LIN {X 0,Y 352.969,Z 845.688,A -85,B 0,C 180,E1 17555.201,E2 17555.201} C_VEL
LIN {X 0,Y 353.121,Z 847.634,A -85,B 0,C 180,E1 17552.272,E2 17552.272} C_VEL
LIN {X 0,Y 353.163,Z 848.054,A -85,B 0,C 180,E1 17549.351,E2 17549.351} C_VEL
LIN {X 0,Y 353.058,Z 846.987,A -85,B 0,C 180,E1 17546.428,E2 17546.428} C_VEL
LIN {X 0,Y 352.892,Z 844.269,A -85,B 0,C 180,E1 17543.493,E2 17543.493} C_VEL
LIN {X 0,Y 352.757,Z 839.752,A -85,B 0,C 180,E1 17540.373,E2 17540.373} C_VEL
LIN {X 0,Y 352.82,Z 833.854,A -85,B 0,C 180,E1 17537.396,E2 17537.396} C_VEL
LIN {X 0,Y 353.289,Z 825.68,A -85,B 0,C 180,E1 17534.205,E2 17534.205} C_VEL
LIN {X 0,Y 354.283,Z 815.339,A -85,B 0,C 180,E1 17530.985,E2 17530.985} C_VEL
LIN {X 0,Y 355.795,Z 803.761,A -85,B 0,C 180,E1 17528.028,E2 17528.028} C_VEL
LIN {X 0,Y 357.865,Z 790.627,A -85,B 0,C 180,E1 17525.223,E2 17525.223} C_VEL
LIN {X 0,Y 360.427,Z 775.886,A -85,B 0,C 180,E1 17522.582,E2 17522.582} C_VEL
LIN {X 0,Y 363.45,Z 759.581,A -85,B 0,C 180,E1 17520.138,E2 17520.138} C_VEL
LIN {X 0,Y 366.634,Z 742.56,A -85,B 0,C 180,E1 17518.009,E2 17518.009} C_VEL
LIN {X 0,Y 369.877,Z 724.753,A -85,B 0,C 180,E1 17516.162,E2 17516.162} C_VEL
LIN {X 0,Y 373,Z 706.679,A -85,B 0,C 180,E1 17514.621,E2 17514.621} C_VEL
LIN {X 0,Y 376.096,Z 686.843,A -85,B 0,C 180,E1 17513.263,E2 17513.263} C_VEL
LIN {X 0,Y 378.966,Z 665.727,A -85,B 0,C 180,E1 17512.158,E2 17512.158} C_VEL
LIN {X 0,Y 381.256,Z 644.268,A -85,B 0,C 180,E1 17511.344,E2 17511.344} C_VEL
LIN {X 0,Y 382.618,Z 622.097,A -85,B 0,C 180,E1 17510.771,E2 17510.771} C_VEL
LIN {X 0,Y 390.111,Z 426.151,A -85,B 0,C 180,E1 17506.792,E2 17506.792} C_VEL
LIN {X 0,Y 386.551,Z 388.013,A -85,B 0,C 180,E1 17505.395,E2 17505.395} C_VEL
LIN {X 0,Y 381.69,Z 378.843,A -85,B 0,C 180,E1 17504.485,E2 17504.485} C_VEL
LIN {X 0,Y 375.097,Z 362.357,A -85,B 0,C 180,E1 17501.725,E2 17501.725} C_VEL
LIN {X 0,Y 367.882,Z 346.536,A -85,B 0,C 180,E1 17498.739,E2 17498.739} C_VEL
LIN {X 0,Y 362.108,Z 334.813,A -85,B 0,C 180,E1 17496.221,E2 17496.221} C_VEL
LIN {X 0,Y 358.372,Z 327.423,A -85,B 0,C 180,E1 17494.497,E2 17494.497} C_VEL
LIN {X 0,Y 355.641,Z 322.528,A -85,B 0,C 180,E1 17493.245,E2 17493.245} C_VEL
LIN {X 0,Y 353.897,Z 318.781,A -85,B 0,C 180,E1 17492.274,E2 17492.274} C_VEL
LIN {X 0,Y 353.829,Z 318.397,A -85,B 0,C 180,E1 17491.709,E2 17491.709} C_VEL
LIN {X 0,Y 353.827,Z 318.394,A -85,B 0,C 180,E1 17487.609,E2 17487.609} C_VEL
LIN {X 0,Y 353.824,Z 318.391,A -85,B 0,C 180,E1 17483.481,E2 17483.481} C_VEL
LIN {X 0,Y 353.819,Z 318.395,A -85,B 0,C 180,E1 17479.478,E2 17479.478} C_VEL
LIN {X 0,Y 353.817,Z 318.407,A -85,B 0,C 180,E1 17475.404,E2 17475.404} C_VEL
LIN {X 0,Y 353.816,Z 318.411,A -85,B 0,C 180,E1 17471.244,E2 17471.244} C_VEL
LIN {X 0,Y 353.812,Z 318.392,A -85,B 0,C 180,E1 17467.142,E2 17467.142} C_VEL
LIN {X 0,Y 353.807,Z 318.384,A -85,B 0,C 180,E1 17463.078,E2 17463.078} C_VEL
LIN {X 0,Y 353.807,Z 318.406,A -85,B 0,C 180,E1 17459.028,E2 17459.028} C_VEL
LIN {X 0,Y 353.816,Z 318.408,A -85,B 0,C 180,E1 17454.811,E2 17454.811} C_VEL
LIN {X 0,Y 353.818,Z 318.382,A -85,B 0,C 180,E1 17450.73,E2 17450.73} C_VEL
LIN {X 0,Y 353.83,Z 318.385,A -85,B 0,C 180,E1 17446.601,E2 17446.601} C_VEL
LIN {X 0,Y 353.845,Z 318.404,A -85,B 0,C 180,E1 17442.401,E2 17442.401} C_VEL
LIN {X 0,Y 353.855,Z 318.406,A -85,B 0,C 180,E1 17438.1,E2 17438.1} C_VEL
LIN {X 0,Y 353.841,Z 318.394,A -85,B 0,C 180,E1 17433.844,E2 17433.844} C_VEL
LIN {X 0,Y 353.843,Z 318.389,A -85,B 0,C 180,E1 17429.802,E2 17429.802} C_VEL
LIN {X 0,Y 353.847,Z 318.389,A -85,B 0,C 180,E1 17425.784,E2 17425.784} C_VEL
LIN {X 0,Y 353.854,Z 318.391,A -85,B 0,C 180,E1 17421.767,E2 17421.767} C_VEL
LIN {X 0,Y 353.858,Z 318.589,A -85,B 0,C 180,E1 17419.146,E2 17419.146} C_VEL
LIN {X 0,Y 355.214,Z 321.938,A -85,B 0,C 180,E1 17418.155,E2 17418.155} C_VEL
LIN {X 0,Y 356.194,Z 323.937,A -85,B 0,C 180,E1 17417.581,E2 17417.581} C_VEL
LIN {X 0,Y 359.806,Z 331.364,A -85,B 0,C 180,E1 17415.55,E2 17415.55} C_VEL
LIN {X 0,Y 365.113,Z 343.733,A -85,B 0,C 180,E1 17412.552,E2 17412.552} C_VEL
LIN {X 0,Y 367.193,Z 348.401,A -85,B 0,C 180,E1 17411.541,E2 17411.541} C_VEL
LIN {X 0,Y 379.033,Z 367.078,A -85,B 0,C 180,E1 17409.324,E2 17409.324} C_VEL
